LIN {X 0,Y 181.648,Z 836.947,A -85,B 0,C 180,E1 -22430.375,E2 -22430.375} C_VEL
LIN {X 0,Y 184.597,Z 832.968,A -85,B 0,C 180,E1 -22433.56,E2 -22433.56} C_VEL
LIN {X 0,Y 188.035,Z 827.945,A -85,B 0,C 180,E1 -22436.645,E2 -22436.645} C_VEL
LIN {X 0,Y 192.221,Z 821.754,A -85,B 0,C 180,E1 -22439.574,E2 -22439.574} C_VEL
LIN {X 0,Y 196.99,Z 814.161,A -85,B 0,C 180,E1 -22442.351,E2 -22442.351} C_VEL
LIN {X 0,Y 201.347,Z 806.526,A -85,B 0,C 180,E1 -22444.553,E2 -22444.553} C_VEL
LIN {X 0,Y 206.537,Z 796.463,A -85,B 0,C 180,E1 -22446.848,E2 -22446.848} C_VEL
LIN {X 0,Y 211.759,Z 785.133,A -85,B 0,C 180,E1 -22448.785,E2 -22448.785} C_VEL
LIN {X 0,Y 216.158,Z 773.945,A -85,B 0,C 180,E1 -22450.253,E2 -22450.253} C_VEL
LIN {X 0,Y 220.233,Z 761.427,A -85,B 0,C 180,E1 -22451.462,E2 -22451.462} C_VEL
LIN {X 0,Y 223.58,Z 747.939,A -85,B 0,C 180,E1 -22452.442,E2 -22452.442} C_VEL
LIN {X 0,Y 226.11,Z 733.339,A -85,B 0,C 180,E1 -22453.139,E2 -22453.139} C_VEL
LIN {X 0,Y 229.571,Z 702.946,A -85,B 0,C 180,E1 -22454.32,E2 -22454.32} C_VEL
LIN {X 0,Y 229.531,Z 699.375,A -85,B 0,C 180,E1 -22454.67,E2 -22454.67} C_VEL
LIN {X 0,Y 226.994,Z 691.679,A -85,B 0,C 180,E1 -22456.697,E2 -22456.697} C_VEL
LIN {X 0,Y 224.698,Z 685.638,A -85,B 0,C 180,E1 -22458.748,E2 -22458.748} C_VEL
LIN {X 0,Y 223.199,Z 682.051,A -85,B 0,C 180,E1 -22460.219,E2 -22460.219} C_VEL
LIN {X 0,Y 221.344,Z 677.62,A -85,B 0,C 180,E1 -22462.368,E2 -22462.368} C_VEL
LIN {X 0,Y 219.109,Z 672.518,A -85,B 0,C 180,E1 -22465.767,E2 -22465.767} C_VEL
LIN {X 0,Y 217.682,Z 669.713,A -85,B 0,C 180,E1 -22469.18,E2 -22469.18} C_VEL
LIN {X 0,Y 217.221,Z 667.959,A -85,B 0,C 180,E1 -22473.066,E2 -22473.066} C_VEL
LIN {X 0,Y 217.771,Z 667.973,A -85,B 0,C 180,E1 -22476.348,E2 -22476.348} C_VEL
LIN {X 0,Y 219.129,Z 668.973,A -85,B 0,C 180,E1 -22479.449,E2 -22479.449} C_VEL
LIN {X 0,Y 221.964,Z 672.987,A -85,B 0,C 180,E1 -22483.528,E2 -22483.528} C_VEL
LIN {X 0,Y 224.726,Z 677.151,A -85,B 0,C 180,E1 -22486.32,E2 -22486.32} C_VEL
LIN {X 0,Y 226.55,Z 680.51,A -85,B 0,C 180,E1 -22487.887,E2 -22487.887} C_VEL
LIN {X 0,Y 230.041,Z 686.961,A -85,B 0,C 180,E1 -22490.49,E2 -22490.49} C_VEL
LIN {X 0,Y 230.883,Z 688.932,A -85,B 0,C 180,E1 -22491.084,E2 -22491.084} C_VEL
LIN {X 0,Y 226.569,Z 725.397,A -85,B 0,C 180,E1 -22492.505,E2 -22492.505} C_VEL
LIN {X 0,Y 224.368,Z 737.74,A -85,B 0,C 180,E1 -22493.254,E2 -22493.254} C_VEL
LIN {X 0,Y 221.212,Z 750.989,A -85,B 0,C 180,E1 -22494.416,E2 -22494.416} C_VEL
LIN {X 0,Y 217.435,Z 762.949,A -85,B 0,C 180,E1 -22495.805,E2 -22495.805} C_VEL
LIN {X 0,Y 212.855,Z 774.862,A -85,B 0,C 180,E1 -22497.634,E2 -22497.634} C_VEL
LIN {X 0,Y 208.036,Z 785.272,A -85,B 0,C 180,E1 -22499.74,E2 -22499.74} C_VEL
LIN {X 0,Y 203.356,Z 793.978,A -85,B 0,C 180,E1 -22501.98,E2 -22501.98} C_VEL
LIN {X 0,Y 198.482,Z 801.986,A -85,B 0,C 180,E1 -22504.581,E2 -22504.581} C_VEL
LIN {X 0,Y 193.325,Z 809.445,A -85,B 0,C 180,E1 -22507.835,E2 -22507.835} C_VEL
LIN {X 0,Y 189.546,Z 814.354,A -85,B 0,C 180,E1 -22510.684,E2 -22510.684} C_VEL
LIN {X 0,Y 185.596,Z 818.913,A -85,B 0,C 180,E1 -22514.249,E2 -22514.249} C_VEL
LIN {X 0,Y 182.384,Z 822.122,A -85,B 0,C 180,E1 -22517.955,E2 -22517.955} C_VEL
LIN {X 0,Y 180.43,Z 823.653,A -85,B 0,C 180,E1 -22520.807,E2 -22520.807} C_VEL
LIN {X 0,Y 178.282,Z 824.713,A -85,B 0,C 180,E1 -22524.957,E2 -22524.957} C_VEL
LIN {X 0,Y 176.87,Z 824.404,A -85,B 0,C 180,E1 -22529.058,E2 -22529.058} C_VEL
LIN {X 0,Y 176.148,Z 822.83,A -85,B 0,C 180,E1 -22533.09,E2 -22533.09} C_VEL
LIN {X 0,Y 176.035,Z 820.076,A -85,B 0,C 180,E1 -22537.02,E2 -22537.02} C_VEL
LIN {X 0,Y 176.43,Z 816.179,A -85,B 0,C 180,E1 -22540.816,E2 -22540.816} C_VEL
LIN {X 0,Y 177.181,Z 811.17,A -85,B 0,C 180,E1 -22544.444,E2 -22544.444} C_VEL
LIN {X 0,Y 178.243,Z 804.98,A -85,B 0,C 180,E1 -22547.914,E2 -22547.914} C_VEL
LIN {X 0,Y 179.786,Z 796.986,A -85,B 0,C 180,E1 -22551.427,E2 -22551.427} C_VEL
LIN {X 0,Y 181.615,Z 788.148,A -85,B 0,C 180,E1 -22554.52,E2 -22554.52} C_VEL
LIN {X 0,Y 183.659,Z 777.988,A -85,B 0,C 180,E1 -22557.337,E2 -22557.337} C_VEL
LIN {X 0,Y 185.886,Z 766.319,A -85,B 0,C 180,E1 -22559.898,E2 -22559.898} C_VEL
LIN {X 0,Y 187.769,Z 754.884,A -85,B 0,C 180,E1 -22561.85,E2 -22561.85} C_VEL
LIN {X 0,Y 189.687,Z 741.422,A -85,B 0,C 180,E1 -22563.605,E2 -22563.605} C_VEL
LIN {X 0,Y 191.005,Z 727.938,A -85,B 0,C 180,E1 -22564.867,E2 -22564.867} C_VEL
LIN {X 0,Y 192.045,Z 714.44,A -85,B 0,C 180,E1 -22565.695,E2 -22565.695} C_VEL
LIN {X 0,Y 195.016,Z 662.361,A -85,B 0,C 180,E1 -22568.021,E2 -22568.021} C_VEL
LIN {X 0,Y 186.643,Z 641.655,A -85,B 0,C 180,E1 -22570.193,E2 -22570.193} C_VEL
LIN {X 0,Y 178.912,Z 624.29,A -85,B 0,C 180,E1 -22572.279,E2 -22572.279} C_VEL
LIN {X 0,Y 178.686,Z 623.228,A -85,B 0,C 180,E1 -22572.403,E2 -22572.403} C_VEL
LIN {X 0,Y 178.894,Z 623.2,A -85,B 0,C 180,E1 -22579.156,E2 -22579.156} C_VEL
LIN {X 0,Y 178.935,Z 623.197,A -85,B 0,C 180,E1 -22583.236,E2 -22583.236} C_VEL
LIN {X 0,Y 179.156,Z 623.169,A -85,B 0,C 180,E1 -22587.754,E2 -22587.754} C_VEL
LIN {X 0,Y 179.371,Z 623.142,A -85,B 0,C 180,E1 -22590.002,E2 -22590.002} C_VEL
LIN {X 0,Y 178.881,Z 623.204,A -85,B 0,C 180,E1 -22594.509,E2 -22594.509} C_VEL
LIN {X 0,Y 178.98,Z 623.19,A -85,B 0,C 180,E1 -22599.039,E2 -22599.039} C_VEL
LIN {X 0,Y 178.684,Z 623.226,A -85,B 0,C 180,E1 -22603.652,E2 -22603.652} C_VEL
LIN {X 0,Y 178.626,Z 623.218,A -85,B 0,C 180,E1 -22609.219,E2 -22609.219} C_VEL
LIN {X 0,Y 178.538,Z 623.247,A -85,B 0,C 180,E1 -22615.127,E2 -22615.127} C_VEL
LIN {X 0,Y 178.505,Z 623.239,A -85,B 0,C 180,E1 -22620.788,E2 -22620.788} C_VEL
LIN {X 0,Y 178.489,Z 623.223,A -85,B 0,C 180,E1 -22624.221,E2 -22624.221} C_VEL
LIN {X 0,Y 178.4,Z 623.256,A -85,B 0,C 180,E1 -22629.076,E2 -22629.076} C_VEL
LIN {X 0,Y 178.412,Z 623.258,A -85,B 0,C 180,E1 -22632.044,E2 -22632.044} C_VEL
LIN {X 0,Y 178.4,Z 623.259,A -85,B 0,C 180,E1 -22635.165,E2 -22635.165} C_VEL
LIN {X 0,Y 178.409,Z 623.246,A -85,B 0,C 180,E1 -22638.461,E2 -22638.461} C_VEL
LIN {X 0,Y 178.428,Z 623.228,A -85,B 0,C 180,E1 -22643.785,E2 -22643.785} C_VEL
LIN {X 0,Y 178.493,Z 623.236,A -85,B 0,C 180,E1 -22646.548,E2 -22646.548} C_VEL
LIN {X 0,Y 178.529,Z 623.245,A -85,B 0,C 180,E1 -22650.008,E2 -22650.008} C_VEL
LIN {X 0,Y 178.526,Z 623.245,A -85,B 0,C 180,E1 -22654.887,E2 -22654.887} C_VEL
LIN {X 0,Y 178.628,Z 623.214,A -85,B 0,C 180,E1 -22660.787,E2 -22660.787} C_VEL
LIN {X 0,Y 178.663,Z 623.21,A -85,B 0,C 180,E1 -22666.349,E2 -22666.349} C_VEL
LIN {X 0,Y 178.919,Z 623.194,A -85,B 0,C 180,E1 -22670.96,E2 -22670.96} C_VEL
LIN {X 0,Y 179.159,Z 623.161,A -85,B 0,C 180,E1 -22677.752,E2 -22677.752} C_VEL
LIN {X 0,Y 179.377,Z 623.123,A -85,B 0,C 180,E1 -22680,E2 -22680} C_VEL
LIN {X 0,Y 178.874,Z 623.193,A -85,B 0,C 180,E1 -22684.507,E2 -22684.507} C_VEL
LIN {X 0,Y 178.919,Z 623.197,A -85,B 0,C 180,E1 -22689.04,E2 -22689.04} C_VEL
LIN {X 0,Y 178.653,Z 623.223,A -85,B 0,C 180,E1 -22693.653,E2 -22693.653} C_VEL
LIN {X 0,Y 178.597,Z 623.239,A -85,B 0,C 180,E1 -22699.185,E2 -22699.185} C_VEL
LIN {X 0,Y 178.527,Z 623.24,A -85,B 0,C 180,E1 -22705.114,E2 -22705.114} C_VEL
LIN {X 0,Y 178.508,Z 623.25,A -85,B 0,C 180,E1 -22710.786,E2 -22710.786} C_VEL
LIN {X 0,Y 178.492,Z 623.248,A -85,B 0,C 180,E1 -22714.219,E2 -22714.219} C_VEL
LIN {X 0,Y 178.402,Z 623.264,A -85,B 0,C 180,E1 -22719.073,E2 -22719.073} C_VEL
LIN {X 0,Y 178.405,Z 623.264,A -85,B 0,C 180,E1 -22722.044,E2 -22722.044} C_VEL
LIN {X 0,Y 178.457,Z 623.395,A -85,B 0,C 180,E1 -22727.484,E2 -22727.484} C_VEL
LIN {X 0,Y 180.474,Z 632.149,A -85,B 0,C 180,E1 -22732.051,E2 -22732.051} C_VEL
LIN {X 0,Y 180.651,Z 633.055,A -85,B 0,C 180,E1 -22732.32,E2 -22732.32} C_VEL
LIN {X 0,Y 188.835,Z 656.224,A -85,B 0,C 180,E1 -22734.741,E2 -22734.741} C_VEL
LIN {X 0,Y 190.706,Z 662.523,A -85,B 0,C 180,E1 -22735.314,E2 -22735.314} C_VEL
LIN {X 0,Y 193.865,Z 696.157,A -85,B 0,C 180,E1 -22737.428,E2 -22737.428} C_VEL
LIN {X 0,Y 191.64,Z 736.563,A -85,B 0,C 180,E1 -22739.265,E2 -22739.265} C_VEL
LIN {X 0,Y 190.442,Z 742.309,A -85,B 0,C 180,E1 -22739.495,E2 -22739.495} C_VEL
LIN {X 0,Y 186.806,Z 751.468,A -85,B 0,C 180,E1 -22739.876,E2 -22739.876} C_VEL
LIN {X 0,Y 183.032,Z 760.446,A -85,B 0,C 180,E1 -22740.48,E2 -22740.48} C_VEL
LIN {X 0,Y 181.66,Z 765.908,A -85,B 0,C 180,E1 -22741.063,E2 -22741.063} C_VEL
LIN {X 0,Y 179.478,Z 778.762,A -85,B 0,C 180,E1 -22742.919,E2 -22742.919} C_VEL
LIN {X 0,Y 177.326,Z 790.159,A -85,B 0,C 180,E1 -22745.093,E2 -22745.093} C_VEL
LIN {X 0,Y 175.234,Z 800.711,A -85,B 0,C 180,E1 -22747.649,E2 -22747.649} C_VEL
LIN {X 0,Y 173.269,Z 809.87,A -85,B 0,C 180,E1 -22750.447,E2 -22750.447} C_VEL
LIN {X 0,Y 171.502,Z 818.953,A -85,B 0,C 180,E1 -22753.94,E2 -22753.94} C_VEL
LIN {X 0,Y 170.239,Z 826.179,A -85,B 0,C 180,E1 -22757.48,E2 -22757.48} C_VEL
LIN {X 0,Y 169.735,Z 831.058,A -85,B 0,C 180,E1 -22760.464,E2 -22760.464} C_VEL
LIN {X 0,Y 169.564,Z 835.798,A -85,B 0,C 180,E1 -22764.125,E2 -22764.125} C_VEL
LIN {X 0,Y 169.464,Z 839.133,A -85,B 0,C 180,E1 -22767.621,E2 -22767.621} C_VEL
LIN {X 0,Y 169.461,Z 840.784,A -85,B 0,C 180,E1 -22769.997,E2 -22769.997} C_VEL
LIN {X 0,Y 169.352,Z 841.973,A -85,B 0,C 180,E1 -22772.376,E2 -22772.376} C_VEL
LIN {X 0,Y 169.192,Z 842.737,A -85,B 0,C 180,E1 -22774.763,E2 -22774.763} C_VEL
LIN {X 0,Y 169.156,Z 843.105,A -85,B 0,C 180,E1 -22777.157,E2 -22777.157} C_VEL
LIN {X 0,Y 169.944,Z 842.621,A -85,B 0,C 180,E1 -22781.931,E2 -22781.931} C_VEL
LIN {X 0,Y 171.776,Z 840.625,A -85,B 0,C 180,E1 -22786.64,E2 -22786.64} C_VEL
LIN {X 0,Y 174.132,Z 838.085,A -85,B 0,C 180,E1 -22790.061,E2 -22790.061} C_VEL
LIN {X 0,Y 176.987,Z 834.626,A -85,B 0,C 180,E1 -22793.394,E2 -22793.394} C_VEL
LIN {X 0,Y 180.46,Z 830.184,A -85,B 0,C 180,E1 -22796.603,E2 -22796.603} C_VEL
LIN {X 0,Y 185.371,Z 823.582,A -85,B 0,C 180,E1 -22800.153,E2 -22800.153} C_VEL
LIN {X 0,Y 191.098,Z 815.187,A -85,B 0,C 180,E1 -22803.478,E2 -22803.478} C_VEL
LIN {X 0,Y 196.603,Z 806.297,A -85,B 0,C 180,E1 -22806.142,E2 -22806.142} C_VEL
LIN {X 0,Y 202.055,Z 796.335,A -85,B 0,C 180,E1 -22808.44,E2 -22808.44} C_VEL
LIN {X 0,Y 207.512,Z 785.05,A -85,B 0,C 180,E1 -22810.367,E2 -22810.367} C_VEL
LIN {X 0,Y 212.688,Z 772.449,A -85,B 0,C 180,E1 -22811.997,E2 -22811.997} C_VEL
LIN {X 0,Y 216.916,Z 759.806,A -85,B 0,C 180,E1 -22813.189,E2 -22813.189} C_VEL
LIN {X 0,Y 220.294,Z 746.746,A -85,B 0,C 180,E1 -22814.094,E2 -22814.094} C_VEL
LIN {X 0,Y 222.866,Z 732.04,A -85,B 0,C 180,E1 -22814.787,E2 -22814.787} C_VEL
LIN {X 0,Y 226.152,Z 704.076,A -85,B 0,C 180,E1 -22815.88,E2 -22815.88} C_VEL
LIN {X 0,Y 225.993,Z 702.661,A -85,B 0,C 180,E1 -22816.101,E2 -22816.101} C_VEL
LIN {X 0,Y 223.948,Z 695.907,A -85,B 0,C 180,E1 -22818.012,E2 -22818.012} C_VEL
LIN {X 0,Y 222.056,Z 690.697,A -85,B 0,C 180,E1 -22819.879,E2 -22819.879} C_VEL
LIN {X 0,Y 219.717,Z 684.472,A -85,B 0,C 180,E1 -22822.696,E2 -22822.696} C_VEL
LIN {X 0,Y 217.5,Z 679.143,A -85,B 0,C 180,E1 -22826.322,E2 -22826.322} C_VEL
LIN {X 0,Y 216.338,Z 676.59,A -85,B 0,C 180,E1 -22829.469,E2 -22829.469} C_VEL
LIN {X 0,Y 215.981,Z 675.016,A -85,B 0,C 180,E1 -22832.899,E2 -22832.899} C_VEL
LIN {X 0,Y 216.492,Z 674.945,A -85,B 0,C 180,E1 -22836.2,E2 -22836.2} C_VEL
LIN {X 0,Y 217.744,Z 675.898,A -85,B 0,C 180,E1 -22839.204,E2 -22839.204} C_VEL
LIN {X 0,Y 220.248,Z 679.639,A -85,B 0,C 180,E1 -22843.065,E2 -22843.065} C_VEL
LIN {X 0,Y 222.809,Z 683.707,A -85,B 0,C 180,E1 -22845.803,E2 -22845.803} C_VEL
LIN {X 0,Y 225.856,Z 689.7,A -85,B 0,C 180,E1 -22848.516,E2 -22848.516} C_VEL
LIN {X 0,Y 227.222,Z 692.457,A -85,B 0,C 180,E1 -22849.602,E2 -22849.602} C_VEL
LIN {X 0,Y 223.019,Z 726.729,A -85,B 0,C 180,E1 -22850.976,E2 -22850.976} C_VEL
LIN {X 0,Y 220.819,Z 738.383,A -85,B 0,C 180,E1 -22851.679,E2 -22851.679} C_VEL
LIN {X 0,Y 217.6,Z 751.285,A -85,B 0,C 180,E1 -22852.81,E2 -22852.81} C_VEL
LIN {X 0,Y 213.823,Z 762.651,A -85,B 0,C 180,E1 -22854.104,E2 -22854.104} C_VEL
LIN {X 0,Y 208.991,Z 774.646,A -85,B 0,C 180,E1 -22855.933,E2 -22855.933} C_VEL
LIN {X 0,Y 204.693,Z 783.723,A -85,B 0,C 180,E1 -22857.689,E2 -22857.689} C_VEL
LIN {X 0,Y 199.568,Z 793.055,A -85,B 0,C 180,E1 -22860,E2 -22860} C_VEL
LIN {X 0,Y 194.308,Z 801.252,A -85,B 0,C 180,E1 -22862.591,E2 -22862.591} C_VEL
LIN {X 0,Y 189.33,Z 808.21,A -85,B 0,C 180,E1 -22865.49,E2 -22865.49} C_VEL
LIN {X 0,Y 184.548,Z 814.138,A -85,B 0,C 180,E1 -22868.762,E2 -22868.762} C_VEL
LIN {X 0,Y 179.974,Z 819.021,A -85,B 0,C 180,E1 -22872.525,E2 -22872.525} C_VEL
LIN {X 0,Y 176.113,Z 822.597,A -85,B 0,C 180,E1 -22876.725,E2 -22876.725} C_VEL
LIN {X 0,Y 173.136,Z 824.6,A -85,B 0,C 180,E1 -22881.001,E2 -22881.001} C_VEL
LIN {X 0,Y 171.005,Z 825.207,A -85,B 0,C 180,E1 -22885.296,E2 -22885.296} C_VEL
LIN {X 0,Y 169.568,Z 824.435,A -85,B 0,C 180,E1 -22889.825,E2 -22889.825} C_VEL
LIN {X 0,Y 168.995,Z 822.592,A -85,B 0,C 180,E1 -22893.727,E2 -22893.727} C_VEL
LIN {X 0,Y 169.023,Z 819.432,A -85,B 0,C 180,E1 -22897.817,E2 -22897.817} C_VEL
LIN {X 0,Y 169.48,Z 815.16,A -85,B 0,C 180,E1 -22901.723,E2 -22901.723} C_VEL
LIN {X 0,Y 170.325,Z 809.758,A -85,B 0,C 180,E1 -22905.46,E2 -22905.46} C_VEL
LIN {X 0,Y 171.522,Z 803.165,A -85,B 0,C 180,E1 -22909.039,E2 -22909.039} C_VEL
LIN {X 0,Y 173.146,Z 795.104,A -85,B 0,C 180,E1 -22912.497,E2 -22912.497} C_VEL
LIN {X 0,Y 175.254,Z 785.219,A -85,B 0,C 180,E1 -22915.849,E2 -22915.849} C_VEL
LIN {X 0,Y 177.249,Z 775.473,A -85,B 0,C 180,E1 -22918.483,E2 -22918.483} C_VEL
LIN {X 0,Y 179.643,Z 763.151,A -85,B 0,C 180,E1 -22921.086,E2 -22921.086} C_VEL
LIN {X 0,Y 181.482,Z 751.827,A -85,B 0,C 180,E1 -22922.96,E2 -22922.96} C_VEL
LIN {X 0,Y 183.261,Z 738.622,A -85,B 0,C 180,E1 -22924.596,E2 -22924.596} C_VEL
LIN {X 0,Y 184.585,Z 724.922,A -85,B 0,C 180,E1 -22925.816,E2 -22925.816} C_VEL
LIN {X 0,Y 185.73,Z 707.38,A -85,B 0,C 180,E1 -22926.761,E2 -22926.761} C_VEL
LIN {X 0,Y 188.344,Z 663.896,A -85,B 0,C 180,E1 -22928.766,E2 -22928.766} C_VEL
LIN {X 0,Y 180.387,Z 644.222,A -85,B 0,C 180,E1 -22930.922,E2 -22930.922} C_VEL
LIN {X 0,Y 172.266,Z 626.336,A -85,B 0,C 180,E1 -22933.199,E2 -22933.199} C_VEL
LIN {X 0,Y 171.62,Z 624.104,A -85,B 0,C 180,E1 -22933.498,E2 -22933.498} C_VEL
LIN {X 0,Y 171.84,Z 624.079,A -85,B 0,C 180,E1 -22938.98,E2 -22938.98} C_VEL
LIN {X 0,Y 171.9,Z 624.074,A -85,B 0,C 180,E1 -22942.957,E2 -22942.957} C_VEL
LIN {X 0,Y 172.103,Z 624.048,A -85,B 0,C 180,E1 -22947.662,E2 -22947.662} C_VEL
LIN {X 0,Y 172.334,Z 624.019,A -85,B 0,C 180,E1 -22950.003,E2 -22950.003} C_VEL
LIN {X 0,Y 171.83,Z 624.083,A -85,B 0,C 180,E1 -22954.695,E2 -22954.695} C_VEL
LIN {X 0,Y 171.912,Z 624.07,A -85,B 0,C 180,E1 -22959.414,E2 -22959.414} C_VEL
LIN {X 0,Y 171.597,Z 624.109,A -85,B 0,C 180,E1 -22964.228,E2 -22964.228} C_VEL
LIN {X 0,Y 171.547,Z 624.098,A -85,B 0,C 180,E1 -22969.564,E2 -22969.564} C_VEL
LIN {X 0,Y 171.473,Z 624.125,A -85,B 0,C 180,E1 -22975.619,E2 -22975.619} C_VEL
LIN {X 0,Y 171.462,Z 624.117,A -85,B 0,C 180,E1 -22980.598,E2 -22980.598} C_VEL
LIN {X 0,Y 171.397,Z 624.109,A -85,B 0,C 180,E1 -22985.037,E2 -22985.037} C_VEL
LIN {X 0,Y 171.362,Z 624.131,A -85,B 0,C 180,E1 -22988.809,E2 -22988.809} C_VEL
LIN {X 0,Y 171.328,Z 624.139,A -85,B 0,C 180,E1 -22994.218,E2 -22994.218} C_VEL
LIN {X 0,Y 171.341,Z 624.123,A -85,B 0,C 180,E1 -22998.983,E2 -22998.983} C_VEL
LIN {X 0,Y 171.392,Z 624.097,A -85,B 0,C 180,E1 -23002.042,E2 -23002.042} C_VEL
LIN {X 0,Y 171.404,Z 624.11,A -85,B 0,C 180,E1 -23005.094,E2 -23005.094} C_VEL
LIN {X 0,Y 171.455,Z 624.124,A -85,B 0,C 180,E1 -23010.536,E2 -23010.536} C_VEL
LIN {X 0,Y 171.451,Z 624.125,A -85,B 0,C 180,E1 -23015.801,E2 -23015.801} C_VEL
LIN {X 0,Y 171.584,Z 624.09,A -85,B 0,C 180,E1 -23020.872,E2 -23020.872} C_VEL
LIN {X 0,Y 171.581,Z 624.087,A -85,B 0,C 180,E1 -23025.773,E2 -23025.773} C_VEL
LIN {X 0,Y 171.855,Z 624.074,A -85,B 0,C 180,E1 -23030.586,E2 -23030.586} C_VEL
LIN {X 0,Y 171.822,Z 624.079,A -85,B 0,C 180,E1 -23035.308,E2 -23035.308} C_VEL
LIN {X 0,Y 172.34,Z 623.998,A -85,B 0,C 180,E1 -23040,E2 -23040} C_VEL
LIN {X 0,Y 171.822,Z 624.072,A -85,B 0,C 180,E1 -23044.693,E2 -23044.693} C_VEL
LIN {X 0,Y 171.856,Z 624.077,A -85,B 0,C 180,E1 -23049.415,E2 -23049.415} C_VEL
LIN {X 0,Y 171.567,Z 624.102,A -85,B 0,C 180,E1 -23054.228,E2 -23054.228} C_VEL
LIN {X 0,Y 171.522,Z 624.12,A -85,B 0,C 180,E1 -23059.533,E2 -23059.533} C_VEL
LIN {X 0,Y 171.466,Z 624.12,A -85,B 0,C 180,E1 -23065.609,E2 -23065.609} C_VEL
LIN {X 0,Y 171.466,Z 624.129,A -85,B 0,C 180,E1 -23070.595,E2 -23070.595} C_VEL
LIN {X 0,Y 171.4,Z 624.136,A -85,B 0,C 180,E1 -23075.034,E2 -23075.034} C_VEL
LIN {X 0,Y 171.364,Z 624.142,A -85,B 0,C 180,E1 -23078.806,E2 -23078.806} C_VEL
LIN {X 0,Y 171.328,Z 624.146,A -85,B 0,C 180,E1 -23084.216,E2 -23084.216} C_VEL
LIN {X 0,Y 171.392,Z 624.272,A -85,B 0,C 180,E1 -23086.817,E2 -23086.817} C_VEL
LIN {X 0,Y 173.24,Z 632.25,A -85,B 0,C 180,E1 -23091.139,E2 -23091.139} C_VEL
LIN {X 0,Y 181.647,Z 655.872,A -85,B 0,C 180,E1 -23093.752,E2 -23093.752} C_VEL
LIN {X 0,Y 184.297,Z 664.633,A -85,B 0,C 180,E1 -23094.603,E2 -23094.603} C_VEL
LIN {X 0,Y 187.221,Z 696.409,A -85,B 0,C 180,E1 -23096.685,E2 -23096.685} C_VEL
LIN {X 0,Y 184.484,Z 742.136,A -85,B 0,C 180,E1 -23098.888,E2 -23098.888} C_VEL
LIN {X 0,Y 183.189,Z 755.342,A -85,B 0,C 180,E1 -23099.922,E2 -23099.922} C_VEL
LIN {X 0,Y 181.66,Z 765.908,A -85,B 0,C 180,E1 -23101.063,E2 -23101.063} C_VEL
LIN {X 0,Y 180.156,Z 771.254,A -85,B 0,C 180,E1 -23101.703,E2 -23101.703} C_VEL
LIN {X 0,Y 175.928,Z 779.57,A -85,B 0,C 180,E1 -23102.786,E2 -23102.786} C_VEL
LIN {X 0,Y 171.556,Z 787.511,A -85,B 0,C 180,E1 -23104.131,E2 -23104.131} C_VEL
LIN {X 0,Y 169.855,Z 792.272,A -85,B 0,C 180,E1 -23105.168,E2 -23105.168} C_VEL
LIN {X 0,Y 167.776,Z 802.309,A -85,B 0,C 180,E1 -23107.849,E2 -23107.849} C_VEL
LIN {X 0,Y 165.879,Z 811.256,A -85,B 0,C 180,E1 -23110.828,E2 -23110.828} C_VEL
LIN {X 0,Y 164.405,Z 818.635,A -85,B 0,C 180,E1 -23113.865,E2 -23113.865} C_VEL
LIN {X 0,Y 163.159,Z 825.839,A -85,B 0,C 180,E1 -23117.56,E2 -23117.56} C_VEL
LIN {X 0,Y 162.576,Z 831.543,A -85,B 0,C 180,E1 -23121.295,E2 -23121.295} C_VEL
LIN {X 0,Y 162.512,Z 835.963,A -85,B 0,C 180,E1 -23125.035,E2 -23125.035} C_VEL
LIN {X 0,Y 162.41,Z 838.219,A -85,B 0,C 180,E1 -23127.517,E2 -23127.517} C_VEL
LIN {X 0,Y 162.397,Z 840.008,A -85,B 0,C 180,E1 -23129.997,E2 -23129.997} C_VEL
LIN {X 0,Y 162.285,Z 841.286,A -85,B 0,C 180,E1 -23132.479,E2 -23132.479} C_VEL
LIN {X 0,Y 162.126,Z 842.116,A -85,B 0,C 180,E1 -23134.971,E2 -23134.971} C_VEL
LIN {X 0,Y 162.396,Z 842.622,A -85,B 0,C 180,E1 -23139.966,E2 -23139.966} C_VEL
LIN {X 0,Y 162.953,Z 842.305,A -85,B 0,C 180,E1 -23142.451,E2 -23142.451} C_VEL
LIN {X 0,Y 164.975,Z 840.477,A -85,B 0,C 180,E1 -23147.347,E2 -23147.347} C_VEL
LIN {X 0,Y 168.35,Z 837.157,A -85,B 0,C 180,E1 -23152.066,E2 -23152.066} C_VEL
LIN {X 0,Y 172.082,Z 833.095,A -85,B 0,C 180,E1 -23155.837,E2 -23155.837} C_VEL
LIN {X 0,Y 176.954,Z 827.175,A -85,B 0,C 180,E1 -23159.763,E2 -23159.763} C_VEL
LIN {X 0,Y 182.672,Z 819.937,A -85,B 0,C 180,E1 -23163.244,E2 -23163.244} C_VEL
LIN {X 0,Y 188.074,Z 812.235,A -85,B 0,C 180,E1 -23166.051,E2 -23166.051} C_VEL
LIN {X 0,Y 194.06,Z 802.72,A -85,B 0,C 180,E1 -23168.658,E2 -23168.658} C_VEL
LIN {X 0,Y 198.865,Z 794.219,A -85,B 0,C 180,E1 -23170.492,E2 -23170.492} C_VEL
LIN {X 0,Y 204.672,Z 782.701,A -85,B 0,C 180,E1 -23172.364,E2 -23172.364} C_VEL
LIN {X 0,Y 209.455,Z 771.196,A -85,B 0,C 180,E1 -23173.789,E2 -23173.789} C_VEL
LIN {X 0,Y 214.151,Z 757.338,A -85,B 0,C 180,E1 -23175.04,E2 -23175.04} C_VEL
LIN {X 0,Y 217.473,Z 744.314,A -85,B 0,C 180,E1 -23175.863,E2 -23175.863} C_VEL
LIN {X 0,Y 219.913,Z 730.436,A -85,B 0,C 180,E1 -23176.497,E2 -23176.497} C_VEL
LIN {X 0,Y 222.876,Z 706.643,A -85,B 0,C 180,E1 -23177.423,E2 -23177.423} C_VEL
LIN {X 0,Y 220.939,Z 700.117,A -85,B 0,C 180,E1 -23179.419,E2 -23179.419} C_VEL
LIN {X 0,Y 219.165,Z 694.647,A -85,B 0,C 180,E1 -23181.566,E2 -23181.566} C_VEL
LIN {X 0,Y 217.607,Z 690.255,A -85,B 0,C 180,E1 -23183.771,E2 -23183.771} C_VEL
LIN {X 0,Y 216.016,Z 685.879,A -85,B 0,C 180,E1 -23186.782,E2 -23186.782} C_VEL
LIN {X 0,Y 214.98,Z 683.376,A -85,B 0,C 180,E1 -23189.928,E2 -23189.928} C_VEL
LIN {X 0,Y 214.743,Z 682.061,A -85,B 0,C 180,E1 -23192.73,E2 -23192.73} C_VEL
LIN {X 0,Y 215.228,Z 681.921,A -85,B 0,C 180,E1 -23196.102,E2 -23196.102} C_VEL
LIN {X 0,Y 216.338,Z 682.759,A -85,B 0,C 180,E1 -23198.895,E2 -23198.895} C_VEL
LIN {X 0,Y 218.64,Z 686.47,A -85,B 0,C 180,E1 -23202.692,E2 -23202.692} C_VEL
LIN {X 0,Y 220.809,Z 690.081,A -85,B 0,C 180,E1 -23205.176,E2 -23205.176} C_VEL
LIN {X 0,Y 223.856,Z 696.508,A -85,B 0,C 180,E1 -23208.093,E2 -23208.093} C_VEL
LIN {X 0,Y 219.867,Z 727.125,A -85,B 0,C 180,E1 -23209.329,E2 -23209.329} C_VEL
LIN {X 0,Y 217.502,Z 739.038,A -85,B 0,C 180,E1 -23210.054,E2 -23210.054} C_VEL
LIN {X 0,Y 214.344,Z 750.993,A -85,B 0,C 180,E1 -23211.084,E2 -23211.084} C_VEL
LIN {X 0,Y 210.603,Z 762.175,A -85,B 0,C 180,E1 -23212.329,E2 -23212.329} C_VEL
LIN {X 0,Y 206.193,Z 772.889,A -85,B 0,C 180,E1 -23213.885,E2 -23213.885} C_VEL
LIN {X 0,Y 200.639,Z 784.1,A -85,B 0,C 180,E1 -23215.983,E2 -23215.983} C_VEL
LIN {X 0,Y 194.872,Z 793.942,A -85,B 0,C 180,E1 -23218.45,E2 -23218.45} C_VEL
LIN {X 0,Y 189.768,Z 801.5,A -85,B 0,C 180,E1 -23220.853,E2 -23220.853} C_VEL
LIN {X 0,Y 184.358,Z 808.629,A -85,B 0,C 180,E1 -23223.825,E2 -23223.825} C_VEL
LIN {X 0,Y 179.771,Z 813.92,A -85,B 0,C 180,E1 -23226.735,E2 -23226.735} C_VEL
LIN {X 0,Y 174.938,Z 818.831,A -85,B 0,C 180,E1 -23230.415,E2 -23230.415} C_VEL
LIN {X 0,Y 170.911,Z 822.338,A -85,B 0,C 180,E1 -23234.283,E2 -23234.283} C_VEL
LIN {X 0,Y 168.679,Z 823.974,A -85,B 0,C 180,E1 -23236.957,E2 -23236.957} C_VEL
LIN {X 0,Y 165.824,Z 825.432,A -85,B 0,C 180,E1 -23241.195,E2 -23241.195} C_VEL
LIN {X 0,Y 163.71,Z 825.596,A -85,B 0,C 180,E1 -23245.648,E2 -23245.648} C_VEL
LIN {X 0,Y 162.396,Z 824.488,A -85,B 0,C 180,E1 -23250.062,E2 -23250.062} C_VEL
LIN {X 0,Y 161.862,Z 822.164,A -85,B 0,C 180,E1 -23254.419,E2 -23254.419} C_VEL
LIN {X 0,Y 161.995,Z 818.668,A -85,B 0,C 180,E1 -23258.66,E2 -23258.66} C_VEL
LIN {X 0,Y 162.574,Z 814.032,A -85,B 0,C 180,E1 -23262.705,E2 -23262.705} C_VEL
LIN {X 0,Y 163.632,Z 807.638,A -85,B 0,C 180,E1 -23266.898,E2 -23266.898} C_VEL
LIN {X 0,Y 164.863,Z 801.169,A -85,B 0,C 180,E1 -23270.254,E2 -23270.254} C_VEL
LIN {X 0,Y 166.691,Z 792.582,A -85,B 0,C 180,E1 -23273.828,E2 -23273.828} C_VEL
LIN {X 0,Y 168.726,Z 783.205,A -85,B 0,C 180,E1 -23276.914,E2 -23276.914} C_VEL
LIN {X 0,Y 170.929,Z 772.602,A -85,B 0,C 180,E1 -23279.705,E2 -23279.705} C_VEL
LIN {X 0,Y 172.995,Z 762.142,A -85,B 0,C 180,E1 -23281.893,E2 -23281.893} C_VEL
LIN {X 0,Y 175.074,Z 749.382,A -85,B 0,C 180,E1 -23283.966,E2 -23283.966} C_VEL
LIN {X 0,Y 176.713,Z 737.201,A -85,B 0,C 180,E1 -23285.461,E2 -23285.461} C_VEL
LIN {X 0,Y 177.996,Z 723.969,A -85,B 0,C 180,E1 -23286.617,E2 -23286.617} C_VEL
LIN {X 0,Y 179.405,Z 703.191,A -85,B 0,C 180,E1 -23287.729,E2 -23287.729} C_VEL
LIN {X 0,Y 181.754,Z 665.678,A -85,B 0,C 180,E1 -23289.525,E2 -23289.525} C_VEL
LIN {X 0,Y 174.275,Z 647.102,A -85,B 0,C 180,E1 -23291.639,E2 -23291.639} C_VEL
LIN {X 0,Y 165.654,Z 627.903,A -85,B 0,C 180,E1 -23294.192,E2 -23294.192} C_VEL
LIN {X 0,Y 164.569,Z 624.982,A -85,B 0,C 180,E1 -23294.601,E2 -23294.601} C_VEL
LIN {X 0,Y 164.85,Z 624.951,A -85,B 0,C 180,E1 -23300.184,E2 -23300.184} C_VEL
LIN {X 0,Y 164.862,Z 624.951,A -85,B 0,C 180,E1 -23302.655,E2 -23302.655} C_VEL
LIN {X 0,Y 165.052,Z 624.926,A -85,B 0,C 180,E1 -23307.562,E2 -23307.562} C_VEL
LIN {X 0,Y 165.297,Z 624.895,A -85,B 0,C 180,E1 -23310.003,E2 -23310.003} C_VEL
LIN {X 0,Y 164.78,Z 624.96,A -85,B 0,C 180,E1 -23314.896,E2 -23314.896} C_VEL
LIN {X 0,Y 164.855,Z 624.949,A -85,B 0,C 180,E1 -23319.821,E2 -23319.821} C_VEL
LIN {X 0,Y 164.539,Z 624.989,A -85,B 0,C 180,E1 -23324.852,E2 -23324.852} C_VEL
LIN {X 0,Y 164.476,Z 624.978,A -85,B 0,C 180,E1 -23329.991,E2 -23329.991} C_VEL
LIN {X 0,Y 164.397,Z 625.006,A -85,B 0,C 180,E1 -23336.136,E2 -23336.136} C_VEL
LIN {X 0,Y 164.392,Z 624.992,A -85,B 0,C 180,E1 -23341.238,E2 -23341.238} C_VEL
LIN {X 0,Y 164.299,Z 625.003,A -85,B 0,C 180,E1 -23346.791,E2 -23346.791} C_VEL
LIN {X 0,Y 164.296,Z 625.015,A -85,B 0,C 180,E1 -23349.918,E2 -23349.918} C_VEL
LIN {X 0,Y 164.284,Z 625.02,A -85,B 0,C 180,E1 -23353.344,E2 -23353.344} C_VEL
LIN {X 0,Y 164.297,Z 625.011,A -85,B 0,C 180,E1 -23356.811,E2 -23356.811} C_VEL
LIN {X 0,Y 164.3,Z 624.992,A -85,B 0,C 180,E1 -23360.354,E2 -23360.354} C_VEL
LIN {X 0,Y 164.336,Z 624.985,A -85,B 0,C 180,E1 -23364.351,E2 -23364.351} C_VEL
LIN {X 0,Y 164.397,Z 625,A -85,B 0,C 180,E1 -23369.136,E2 -23369.136} C_VEL
LIN {X 0,Y 164.413,Z 625.003,A -85,B 0,C 180,E1 -23374.694,E2 -23374.694} C_VEL
LIN {X 0,Y 164.491,Z 624.975,A -85,B 0,C 180,E1 -23380.053,E2 -23380.053} C_VEL
LIN {X 0,Y 164.511,Z 624.964,A -85,B 0,C 180,E1 -23385.148,E2 -23385.148} C_VEL
LIN {X 0,Y 164.775,Z 624.955,A -85,B 0,C 180,E1 -23390.177,E2 -23390.177} C_VEL
LIN {X 0,Y 164.838,Z 624.95,A -85,B 0,C 180,E1 -23392.652,E2 -23392.652} C_VEL
LIN {X 0,Y 165.055,Z 624.918,A -85,B 0,C 180,E1 -23397.56,E2 -23397.56} C_VEL
LIN {X 0,Y 165.302,Z 624.874,A -85,B 0,C 180,E1 -23400,E2 -23400} C_VEL
LIN {X 0,Y 164.771,Z 624.951,A -85,B 0,C 180,E1 -23404.894,E2 -23404.894} C_VEL
LIN {X 0,Y 164.839,Z 624.949,A -85,B 0,C 180,E1 -23407.349,E2 -23407.349} C_VEL
LIN {X 0,Y 164.71,Z 624.965,A -85,B 0,C 180,E1 -23411.061,E2 -23411.061} C_VEL
LIN {X 0,Y 164.46,Z 624.995,A -85,B 0,C 180,E1 -23417.406,E2 -23417.406} C_VEL
LIN {X 0,Y 164.456,Z 625.001,A -85,B 0,C 180,E1 -23419.992,E2 -23419.992} C_VEL
LIN {X 0,Y 164.393,Z 625.001,A -85,B 0,C 180,E1 -23426.128,E2 -23426.128} C_VEL
LIN {X 0,Y 164.396,Z 625.006,A -85,B 0,C 180,E1 -23431.235,E2 -23431.235} C_VEL
LIN {X 0,Y 164.301,Z 625.019,A -85,B 0,C 180,E1 -23436.788,E2 -23436.788} C_VEL
LIN {X 0,Y 164.297,Z 625.021,A -85,B 0,C 180,E1 -23439.915,E2 -23439.915} C_VEL
LIN {X 0,Y 164.288,Z 625.024,A -85,B 0,C 180,E1 -23444.897,E2 -23444.897} C_VEL
LIN {X 0,Y 164.337,Z 625.089,A -85,B 0,C 180,E1 -23446.082,E2 -23446.082} C_VEL
LIN {X 0,Y 165.907,Z 631.794,A -85,B 0,C 180,E1 -23449.914,E2 -23449.914} C_VEL
LIN {X 0,Y 174.901,Z 656.794,A -85,B 0,C 180,E1 -23452.854,E2 -23452.854} C_VEL
LIN {X 0,Y 177.785,Z 665.671,A -85,B 0,C 180,E1 -23453.773,E2 -23453.773} C_VEL
LIN {X 0,Y 180.611,Z 696.413,A -85,B 0,C 180,E1 -23455.882,E2 -23455.882} C_VEL
LIN {X 0,Y 177.779,Z 741.96,A -85,B 0,C 180,E1 -23458.16,E2 -23458.16} C_VEL
LIN {X 0,Y 176.362,Z 755.741,A -85,B 0,C 180,E1 -23459.295,E2 -23459.295} C_VEL
LIN {X 0,Y 174.452,Z 768.195,A -85,B 0,C 180,E1 -23460.757,E2 -23460.757} C_VEL
LIN {X 0,Y 172.23,Z 780.264,A -85,B 0,C 180,E1 -23462.67,E2 -23462.67} C_VEL
LIN {X 0,Y 170.078,Z 791.308,A -85,B 0,C 180,E1 -23464.938,E2 -23464.938} C_VEL
LIN {X 0,Y 169.855,Z 792.272,A -85,B 0,C 180,E1 -23465.168,E2 -23465.168} C_VEL
LIN {X 0,Y 168.17,Z 796.897,A -85,B 0,C 180,E1 -23466.293,E2 -23466.293} C_VEL
LIN {X 0,Y 163.831,Z 803.893,A -85,B 0,C 180,E1 -23468.206,E2 -23468.206} C_VEL
LIN {X 0,Y 159.597,Z 810.395,A -85,B 0,C 180,E1 -23470.404,E2 -23470.404} C_VEL
LIN {X 0,Y 158.11,Z 814.21,A -85,B 0,C 180,E1 -23471.939,E2 -23471.939} C_VEL
LIN {X 0,Y 156.601,Z 822.119,A -85,B 0,C 180,E1 -23475.707,E2 -23475.707} C_VEL
LIN {X 0,Y 155.719,Z 828.51,A -85,B 0,C 180,E1 -23479.597,E2 -23479.597} C_VEL
LIN {X 0,Y 155.439,Z 834.189,A -85,B 0,C 180,E1 -23484.107,E2 -23484.107} C_VEL
LIN {X 0,Y 155.359,Z 837.282,A -85,B 0,C 180,E1 -23487.404,E2 -23487.404} C_VEL
LIN {X 0,Y 155.342,Z 839.144,A -85,B 0,C 180,E1 -23489.997,E2 -23489.997} C_VEL
LIN {X 0,Y 155.22,Z 840.542,A -85,B 0,C 180,E1 -23492.592,E2 -23492.592} C_VEL
LIN {X 0,Y 155.046,Z 841.481,A -85,B 0,C 180,E1 -23495.199,E2 -23495.199} C_VEL
LIN {X 0,Y 155.388,Z 842.15,A -85,B 0,C 180,E1 -23500.42,E2 -23500.42} C_VEL
LIN {X 0,Y 156.87,Z 841.331,A -85,B 0,C 180,E1 -23505.59,E2 -23505.59} C_VEL
LIN {X 0,Y 159.879,Z 838.979,A -85,B 0,C 180,E1 -23510.586,E2 -23510.586} C_VEL
LIN {X 0,Y 164.048,Z 835.058,A -85,B 0,C 180,E1 -23515.364,E2 -23515.364} C_VEL
LIN {X 0,Y 167.907,Z 831.031,A -85,B 0,C 180,E1 -23518.77,E2 -23518.77} C_VEL
LIN {X 0,Y 172.46,Z 825.955,A -85,B 0,C 180,E1 -23521.987,E2 -23521.987} C_VEL
LIN {X 0,Y 178.589,Z 818.53,A -85,B 0,C 180,E1 -23525.479,E2 -23525.479} C_VEL
LIN {X 0,Y 184.463,Z 810.644,A -85,B 0,C 180,E1 -23528.249,E2 -23528.249} C_VEL
LIN {X 0,Y 190.857,Z 801.001,A -85,B 0,C 180,E1 -23530.811,E2 -23530.811} C_VEL
LIN {X 0,Y 196.599,Z 791.168,A -85,B 0,C 180,E1 -23532.779,E2 -23532.779} C_VEL
LIN {X 0,Y 202.675,Z 778.963,A -85,B 0,C 180,E1 -23534.6,E2 -23534.6} C_VEL
LIN {X 0,Y 207.748,Z 766.798,A -85,B 0,C 180,E1 -23535.958,E2 -23535.958} C_VEL
LIN {X 0,Y 212.093,Z 753.545,A -85,B 0,C 180,E1 -23537.034,E2 -23537.034} C_VEL
LIN {X 0,Y 215.479,Z 739.849,A -85,B 0,C 180,E1 -23537.803,E2 -23537.803} C_VEL
LIN {X 0,Y 218.315,Z 720.921,A -85,B 0,C 180,E1 -23538.564,E2 -23538.564} C_VEL
LIN {X 0,Y 219.717,Z 709.868,A -85,B 0,C 180,E1 -23539.011,E2 -23539.011} C_VEL
LIN {X 0,Y 217.893,Z 703.232,A -85,B 0,C 180,E1 -23541.3,E2 -23541.3} C_VEL
LIN {X 0,Y 216.639,Z 699.413,A -85,B 0,C 180,E1 -23543.019,E2 -23543.019} C_VEL
LIN {X 0,Y 215.773,Z 696.529,A -85,B 0,C 180,E1 -23544.543,E2 -23544.543} C_VEL
LIN {X 0,Y 214.526,Z 692.552,A -85,B 0,C 180,E1 -23547.294,E2 -23547.294} C_VEL
LIN {X 0,Y 213.681,Z 690.279,A -85,B 0,C 180,E1 -23550.205,E2 -23550.205} C_VEL
LIN {X 0,Y 213.522,Z 688.933,A -85,B 0,C 180,E1 -23553.444,E2 -23553.444} C_VEL
LIN {X 0,Y 214.318,Z 689.078,A -85,B 0,C 180,E1 -23557.134,E2 -23557.134} C_VEL
LIN {X 0,Y 215.11,Z 690.06,A -85,B 0,C 180,E1 -23559.046,E2 -23559.046} C_VEL
LIN {X 0,Y 216.943,Z 693.058,A -85,B 0,C 180,E1 -23562.164,E2 -23562.164} C_VEL
LIN {X 0,Y 218.934,Z 696.625,A -85,B 0,C 180,E1 -23564.645,E2 -23564.645} C_VEL
LIN {X 0,Y 220.653,Z 700.602,A -85,B 0,C 180,E1 -23566.545,E2 -23566.545} C_VEL
LIN {X 0,Y 216.893,Z 728.131,A -85,B 0,C 180,E1 -23567.662,E2 -23567.662} C_VEL
LIN {X 0,Y 214.085,Z 741.371,A -85,B 0,C 180,E1 -23568.479,E2 -23568.479} C_VEL
LIN {X 0,Y 210.655,Z 753.344,A -85,B 0,C 180,E1 -23569.548,E2 -23569.548} C_VEL
LIN {X 0,Y 206.43,Z 764.7,A -85,B 0,C 180,E1 -23570.849,E2 -23570.849} C_VEL
LIN {X 0,Y 201.637,Z 775.401,A -85,B 0,C 180,E1 -23572.475,E2 -23572.475} C_VEL
LIN {X 0,Y 195.817,Z 786.26,A -85,B 0,C 180,E1 -23574.594,E2 -23574.594} C_VEL
LIN {X 0,Y 190.01,Z 795.516,A -85,B 0,C 180,E1 -23576.986,E2 -23576.986} C_VEL
LIN {X 0,Y 184.54,Z 802.988,A -85,B 0,C 180,E1 -23579.454,E2 -23579.454} C_VEL
LIN {X 0,Y 179.236,Z 809.433,A -85,B 0,C 180,E1 -23582.247,E2 -23582.247} C_VEL
LIN {X 0,Y 173.438,Z 815.572,A -85,B 0,C 180,E1 -23585.814,E2 -23585.814} C_VEL
LIN {X 0,Y 168.396,Z 820.168,A -85,B 0,C 180,E1 -23589.61,E2 -23589.61} C_VEL
LIN {X 0,Y 165.43,Z 822.504,A -85,B 0,C 180,E1 -23592.295,E2 -23592.295} C_VEL
LIN {X 0,Y 161.508,Z 825.003,A -85,B 0,C 180,E1 -23596.809,E2 -23596.809} C_VEL
LIN {X 0,Y 158.506,Z 826.1,A -85,B 0,C 180,E1 -23601.398,E2 -23601.398} C_VEL
LIN {X 0,Y 156.422,Z 825.868,A -85,B 0,C 180,E1 -23606.033,E2 -23606.033} C_VEL
LIN {X 0,Y 155.181,Z 824.351,A -85,B 0,C 180,E1 -23610.634,E2 -23610.634} C_VEL
LIN {X 0,Y 154.759,Z 821.612,A -85,B 0,C 180,E1 -23615.178,E2 -23615.178} C_VEL
LIN {X 0,Y 154.963,Z 817.723,A -85,B 0,C 180,E1 -23619.561,E2 -23619.561} C_VEL
LIN {X 0,Y 155.709,Z 812.68,A -85,B 0,C 180,E1 -23623.771,E2 -23623.771} C_VEL
LIN {X 0,Y 156.776,Z 806.512,A -85,B 0,C 180,E1 -23627.75,E2 -23627.75} C_VEL
LIN {X 0,Y 158.281,Z 798.984,A -85,B 0,C 180,E1 -23631.569,E2 -23631.569} C_VEL
LIN {X 0,Y 160.332,Z 789.805,A -85,B 0,C 180,E1 -23635.264,E2 -23635.264} C_VEL
LIN {X 0,Y 162.446,Z 780.34,A -85,B 0,C 180,E1 -23638.279,E2 -23638.279} C_VEL
LIN {X 0,Y 164.688,Z 769.498,A -85,B 0,C 180,E1 -23641.024,E2 -23641.024} C_VEL
LIN {X 0,Y 167.005,Z 757.465,A -85,B 0,C 180,E1 -23643.412,E2 -23643.412} C_VEL
LIN {X 0,Y 169.004,Z 744.872,A -85,B 0,C 180,E1 -23645.304,E2 -23645.304} C_VEL
LIN {X 0,Y 170.651,Z 731.287,A -85,B 0,C 180,E1 -23646.811,E2 -23646.811} C_VEL
LIN {X 0,Y 171.868,Z 717.051,A -85,B 0,C 180,E1 -23647.84,E2 -23647.84} C_VEL
LIN {X 0,Y 175.082,Z 667.143,A -85,B 0,C 180,E1 -23650.34,E2 -23650.34} C_VEL
LIN {X 0,Y 166.978,Z 647.126,A -85,B 0,C 180,E1 -23652.775,E2 -23652.775} C_VEL
LIN {X 0,Y 158.692,Z 628.928,A -85,B 0,C 180,E1 -23655.366,E2 -23655.366} C_VEL
LIN {X 0,Y 157.651,Z 626.528,A -85,B 0,C 180,E1 -23655.721,E2 -23655.721} C_VEL
LIN {X 0,Y 157.538,Z 625.861,A -85,B 0,C 180,E1 -23655.801,E2 -23655.801} C_VEL
LIN {X 0,Y 157.768,Z 625.832,A -85,B 0,C 180,E1 -23659.739,E2 -23659.739} C_VEL
LIN {X 0,Y 157.824,Z 625.827,A -85,B 0,C 180,E1 -23662.326,E2 -23662.326} C_VEL
LIN {X 0,Y 158.259,Z 625.772,A -85,B 0,C 180,E1 -23670.003,E2 -23670.003} C_VEL
LIN {X 0,Y 157.827,Z 625.823,A -85,B 0,C 180,E1 -23677.68,E2 -23677.68} C_VEL
LIN {X 0,Y 157.707,Z 625.837,A -85,B 0,C 180,E1 -23681.364,E2 -23681.364} C_VEL
LIN {X 0,Y 157.465,Z 625.868,A -85,B 0,C 180,E1 -23685.536,E2 -23685.536} C_VEL
LIN {X 0,Y 157.373,Z 625.866,A -85,B 0,C 180,E1 -23690.935,E2 -23690.935} C_VEL
LIN {X 0,Y 157.319,Z 625.889,A -85,B 0,C 180,E1 -23696.688,E2 -23696.688} C_VEL
LIN {X 0,Y 157.285,Z 625.87,A -85,B 0,C 180,E1 -23702.428,E2 -23702.428} C_VEL
LIN {X 0,Y 157.272,Z 625.876,A -85,B 0,C 180,E1 -23706.452,E2 -23706.452} C_VEL
LIN {X 0,Y 157.215,Z 625.898,A -85,B 0,C 180,E1 -23712.113,E2 -23712.113} C_VEL
LIN {X 0,Y 157.216,Z 625.885,A -85,B 0,C 180,E1 -23717.891,E2 -23717.891} C_VEL
LIN {X 0,Y 157.273,Z 625.856,A -85,B 0,C 180,E1 -23723.552,E2 -23723.552} C_VEL
LIN {X 0,Y 157.3,Z 625.881,A -85,B 0,C 180,E1 -23728.097,E2 -23728.097} C_VEL
LIN {X 0,Y 157.322,Z 625.889,A -85,B 0,C 180,E1 -23733.466,E2 -23733.466} C_VEL
LIN {X 0,Y 157.398,Z 625.86,A -85,B 0,C 180,E1 -23739.671,E2 -23739.671} C_VEL
LIN {X 0,Y 157.447,Z 625.837,A -85,B 0,C 180,E1 -23744.466,E2 -23744.466} C_VEL
LIN {X 0,Y 157.697,Z 625.834,A -85,B 0,C 180,E1 -23749.732,E2 -23749.732} C_VEL
LIN {X 0,Y 157.775,Z 625.831,A -85,B 0,C 180,E1 -23752.321,E2 -23752.321} C_VEL
LIN {X 0,Y 158.265,Z 625.749,A -85,B 0,C 180,E1 -23760,E2 -23760} C_VEL
LIN {X 0,Y 157.775,Z 625.829,A -85,B 0,C 180,E1 -23767.68,E2 -23767.68} C_VEL
LIN {X 0,Y 157.641,Z 625.846,A -85,B 0,C 180,E1 -23771.23,E2 -23771.23} C_VEL
LIN {X 0,Y 157.429,Z 625.86,A -85,B 0,C 180,E1 -23775.537,E2 -23775.537} C_VEL
LIN {X 0,Y 157.364,Z 625.886,A -85,B 0,C 180,E1 -23780.934,E2 -23780.934} C_VEL
LIN {X 0,Y 157.316,Z 625.885,A -85,B 0,C 180,E1 -23786.68,E2 -23786.68} C_VEL
LIN {X 0,Y 157.288,Z 625.889,A -85,B 0,C 180,E1 -23792.425,E2 -23792.425} C_VEL
LIN {X 0,Y 157.275,Z 625.894,A -85,B 0,C 180,E1 -23796.448,E2 -23796.448} C_VEL
LIN {X 0,Y 157.217,Z 625.904,A -85,B 0,C 180,E1 -23802.109,E2 -23802.109} C_VEL
LIN {X 0,Y 157.281,Z 625.967,A -85,B 0,C 180,E1 -23805.35,E2 -23805.35} C_VEL
LIN {X 0,Y 158.497,Z 631.34,A -85,B 0,C 180,E1 -23808.576,E2 -23808.576} C_VEL
LIN {X 0,Y 166.387,Z 652.552,A -85,B 0,C 180,E1 -23811.299,E2 -23811.299} C_VEL
LIN {X 0,Y 171.371,Z 668.004,A -85,B 0,C 180,E1 -23813.013,E2 -23813.013} C_VEL
LIN {X 0,Y 173.975,Z 696.993,A -85,B 0,C 180,E1 -23815.084,E2 -23815.084} C_VEL
LIN {X 0,Y 171.123,Z 741.157,A -85,B 0,C 180,E1 -23817.379,E2 -23817.379} C_VEL
LIN {X 0,Y 169.734,Z 754.327,A -85,B 0,C 180,E1 -23818.48,E2 -23818.48} C_VEL
LIN {X 0,Y 167.95,Z 766.06,A -85,B 0,C 180,E1 -23819.855,E2 -23819.855} C_VEL
LIN {X 0,Y 165.669,Z 778.535,A -85,B 0,C 180,E1 -23821.837,E2 -23821.837} C_VEL
LIN {X 0,Y 163.403,Z 789.798,A -85,B 0,C 180,E1 -23824.181,E2 -23824.181} C_VEL
LIN {X 0,Y 161.207,Z 800.063,A -85,B 0,C 180,E1 -23826.895,E2 -23826.895} C_VEL
LIN {X 0,Y 159.154,Z 809.302,A -85,B 0,C 180,E1 -23829.985,E2 -23829.985} C_VEL
LIN {X 0,Y 158.11,Z 814.21,A -85,B 0,C 180,E1 -23831.939,E2 -23831.939} C_VEL
LIN {X 0,Y 156.689,Z 817.844,A -85,B 0,C 180,E1 -23833.559,E2 -23833.559} C_VEL
LIN {X 0,Y 152.862,Z 823.049,A -85,B 0,C 180,E1 -23836.347,E2 -23836.347} C_VEL
LIN {X 0,Y 149.356,Z 827.666,A -85,B 0,C 180,E1 -23839.425,E2 -23839.425} C_VEL
LIN {X 0,Y 148.465,Z 830.248,A -85,B 0,C 180,E1 -23841.441,E2 -23841.441} C_VEL
LIN {X 0,Y 148.379,Z 834.525,A -85,B 0,C 180,E1 -23845.272,E2 -23845.272} C_VEL
LIN {X 0,Y 148.31,Z 836.308,A -85,B 0,C 180,E1 -23847.281,E2 -23847.281} C_VEL
LIN {X 0,Y 148.288,Z 838.264,A -85,B 0,C 180,E1 -23849.997,E2 -23849.997} C_VEL
LIN {X 0,Y 148.067,Z 840.513,A -85,B 0,C 180,E1 -23854.605,E2 -23854.605} C_VEL
LIN {X 0,Y 148.007,Z 841.435,A -85,B 0,C 180,E1 -23858.187,E2 -23858.187} C_VEL
LIN {X 0,Y 149.034,Z 841.536,A -85,B 0,C 180,E1 -23863.635,E2 -23863.635} C_VEL
LIN {X 0,Y 151.444,Z 840.168,A -85,B 0,C 180,E1 -23868.953,E2 -23868.953} C_VEL
LIN {X 0,Y 155.253,Z 837.305,A -85,B 0,C 180,E1 -23874.039,E2 -23874.039} C_VEL
LIN {X 0,Y 160.304,Z 832.824,A -85,B 0,C 180,E1 -23878.83,E2 -23878.83} C_VEL
LIN {X 0,Y 164.831,Z 828.322,A -85,B 0,C 180,E1 -23882.203,E2 -23882.203} C_VEL
LIN {X 0,Y 171.089,Z 821.734,A -85,B 0,C 180,E1 -23885.825,E2 -23885.825} C_VEL
LIN {X 0,Y 176.963,Z 814.702,A -85,B 0,C 180,E1 -23888.716,E2 -23888.716} C_VEL
LIN {X 0,Y 183.408,Z 806.054,A -85,B 0,C 180,E1 -23891.373,E2 -23891.373} C_VEL
LIN {X 0,Y 189.129,Z 797.437,A -85,B 0,C 180,E1 -23893.426,E2 -23893.426} C_VEL
LIN {X 0,Y 195.294,Z 786.992,A -85,B 0,C 180,E1 -23895.292,E2 -23895.292} C_VEL
LIN {X 0,Y 201.042,Z 775.39,A -85,B 0,C 180,E1 -23896.862,E2 -23896.862} C_VEL
LIN {X 0,Y 205.733,Z 764.035,A -85,B 0,C 180,E1 -23897.984,E2 -23897.984} C_VEL
LIN {X 0,Y 209.903,Z 751.267,A -85,B 0,C 180,E1 -23898.957,E2 -23898.957} C_VEL
LIN {X 0,Y 213.219,Z 737.653,A -85,B 0,C 180,E1 -23899.674,E2 -23899.674} C_VEL
LIN {X 0,Y 216.764,Z 714.225,A -85,B 0,C 180,E1 -23900.567,E2 -23900.567} C_VEL
LIN {X 0,Y 216.803,Z 713.203,A -85,B 0,C 180,E1 -23900.685,E2 -23900.685} C_VEL
LIN {X 0,Y 215.285,Z 707.337,A -85,B 0,C 180,E1 -23902.917,E2 -23902.917} C_VEL
LIN {X 0,Y 214.082,Z 703.019,A -85,B 0,C 180,E1 -23905.152,E2 -23905.152} C_VEL
LIN {X 0,Y 213.063,Z 699.275,A -85,B 0,C 180,E1 -23907.762,E2 -23907.762} C_VEL
LIN {X 0,Y 212.375,Z 697.166,A -85,B 0,C 180,E1 -23910.511,E2 -23910.511} C_VEL
LIN {X 0,Y 212.26,Z 695.947,A -85,B 0,C 180,E1 -23913.372,E2 -23913.372} C_VEL
LIN {X 0,Y 212.88,Z 695.949,A -85,B 0,C 180,E1 -23916.661,E2 -23916.661} C_VEL
LIN {X 0,Y 213.651,Z 696.819,A -85,B 0,C 180,E1 -23918.617,E2 -23918.617} C_VEL
LIN {X 0,Y 215.342,Z 699.819,A -85,B 0,C 180,E1 -23921.753,E2 -23921.753} C_VEL
LIN {X 0,Y 217.094,Z 703.273,A -85,B 0,C 180,E1 -23924.141,E2 -23924.141} C_VEL
LIN {X 0,Y 217.769,Z 705.006,A -85,B 0,C 180,E1 -23924.964,E2 -23924.964} C_VEL
LIN {X 0,Y 214.289,Z 728.814,A -85,B 0,C 180,E1 -23925.919,E2 -23925.919} C_VEL
LIN {X 0,Y 211.456,Z 741.514,A -85,B 0,C 180,E1 -23926.691,E2 -23926.691} C_VEL
LIN {X 0,Y 208.202,Z 752.451,A -85,B 0,C 180,E1 -23927.625,E2 -23927.625} C_VEL
LIN {X 0,Y 203.405,Z 765.104,A -85,B 0,C 180,E1 -23929.045,E2 -23929.045} C_VEL
LIN {X 0,Y 197.877,Z 776.861,A -85,B 0,C 180,E1 -23930.802,E2 -23930.802} C_VEL
LIN {X 0,Y 192.009,Z 787.088,A -85,B 0,C 180,E1 -23932.817,E2 -23932.817} C_VEL
LIN {X 0,Y 186.07,Z 795.975,A -85,B 0,C 180,E1 -23935.125,E2 -23935.125} C_VEL
LIN {X 0,Y 179.917,Z 803.948,A -85,B 0,C 180,E1 -23937.761,E2 -23937.761} C_VEL
LIN {X 0,Y 173.216,Z 811.412,A -85,B 0,C 180,E1 -23941.162,E2 -23941.162} C_VEL
LIN {X 0,Y 167.163,Z 817.188,A -85,B 0,C 180,E1 -23944.823,E2 -23944.823} C_VEL
LIN {X 0,Y 161.816,Z 821.529,A -85,B 0,C 180,E1 -23948.782,E2 -23948.782} C_VEL
LIN {X 0,Y 157.462,Z 824.414,A -85,B 0,C 180,E1 -23952.895,E2 -23952.895} C_VEL
LIN {X 0,Y 154.181,Z 826.003,A -85,B 0,C 180,E1 -23956.827,E2 -23956.827} C_VEL
LIN {X 0,Y 151.06,Z 826.627,A -85,B 0,C 180,E1 -23961.851,E2 -23961.851} C_VEL
LIN {X 0,Y 149.13,Z 825.964,A -85,B 0,C 180,E1 -23966.447,E2 -23966.447} C_VEL
LIN {X 0,Y 147.935,Z 823.936,A -85,B 0,C 180,E1 -23971.505,E2 -23971.505} C_VEL
LIN {X 0,Y 147.669,Z 820.942,A -85,B 0,C 180,E1 -23976,E2 -23976} C_VEL
LIN {X 0,Y 148.003,Z 816.642,A -85,B 0,C 180,E1 -23980.561,E2 -23980.561} C_VEL
LIN {X 0,Y 148.901,Z 810.964,A -85,B 0,C 180,E1 -23985.071,E2 -23985.071} C_VEL
LIN {X 0,Y 150.062,Z 804.584,A -85,B 0,C 180,E1 -23989.033,E2 -23989.033} C_VEL
LIN {X 0,Y 151.766,Z 796.547,A -85,B 0,C 180,E1 -23992.99,E2 -23992.99} C_VEL
LIN {X 0,Y 154.07,Z 786.649,A -85,B 0,C 180,E1 -23996.816,E2 -23996.816} C_VEL
LIN {X 0,Y 156.224,Z 777.046,A -85,B 0,C 180,E1 -23999.769,E2 -23999.769} C_VEL
LIN {X 0,Y 158.571,Z 766.107,A -85,B 0,C 180,E1 -24002.426,E2 -24002.426} C_VEL
LIN {X 0,Y 160.714,Z 754.518,A -85,B 0,C 180,E1 -24004.645,E2 -24004.645} C_VEL
LIN {X 0,Y 162.653,Z 742.455,A -85,B 0,C 180,E1 -24006.412,E2 -24006.412} C_VEL
LIN {X 0,Y 164.254,Z 728.323,A -85,B 0,C 180,E1 -24007.907,E2 -24007.907} C_VEL
LIN {X 0,Y 165.4,Z 715.017,A -85,B 0,C 180,E1 -24008.812,E2 -24008.812} C_VEL
LIN {X 0,Y 168.446,Z 668.634,A -85,B 0,C 180,E1 -24011.218,E2 -24011.218} C_VEL
LIN {X 0,Y 160.781,Z 649.862,A -85,B 0,C 180,E1 -24013.611,E2 -24013.611} C_VEL
LIN {X 0,Y 153.53,Z 633.685,A -85,B 0,C 180,E1 -24016.013,E2 -24016.013} C_VEL
LIN {X 0,Y 150.664,Z 627.552,A -85,B 0,C 180,E1 -24017.005,E2 -24017.005} C_VEL
LIN {X 0,Y 150.545,Z 626.732,A -85,B 0,C 180,E1 -24017.144,E2 -24017.144} C_VEL
LIN {X 0,Y 150.762,Z 626.706,A -85,B 0,C 180,E1 -24021.964,E2 -24021.964} C_VEL
LIN {X 0,Y 151.22,Z 626.649,A -85,B 0,C 180,E1 -24030.003,E2 -24030.003} C_VEL
LIN {X 0,Y 150.765,Z 626.703,A -85,B 0,C 180,E1 -24038.042,E2 -24038.042} C_VEL
LIN {X 0,Y 150.637,Z 626.717,A -85,B 0,C 180,E1 -24041.548,E2 -24041.548} C_VEL
LIN {X 0,Y 150.371,Z 626.752,A -85,B 0,C 180,E1 -24046.289,E2 -24046.289} C_VEL
LIN {X 0,Y 150.354,Z 626.739,A -85,B 0,C 180,E1 -24050.795,E2 -24050.795} C_VEL
LIN {X 0,Y 150.249,Z 626.768,A -85,B 0,C 180,E1 -24057.286,E2 -24057.286} C_VEL
LIN {X 0,Y 150.224,Z 626.746,A -85,B 0,C 180,E1 -24062.638,E2 -24062.638} C_VEL
LIN {X 0,Y 150.177,Z 626.764,A -85,B 0,C 180,E1 -24067.476,E2 -24067.476} C_VEL
LIN {X 0,Y 150.155,Z 626.78,A -85,B 0,C 180,E1 -24071.507,E2 -24071.507} C_VEL
LIN {X 0,Y 150.13,Z 626.777,A -85,B 0,C 180,E1 -24075.397,E2 -24075.397} C_VEL
LIN {X 0,Y 150.155,Z 626.758,A -85,B 0,C 180,E1 -24079.06,E2 -24079.06} C_VEL
LIN {X 0,Y 150.184,Z 626.734,A -85,B 0,C 180,E1 -24082.71,E2 -24082.71} C_VEL
LIN {X 0,Y 150.221,Z 626.757,A -85,B 0,C 180,E1 -24087.369,E2 -24087.369} C_VEL
LIN {X 0,Y 150.247,Z 626.768,A -85,B 0,C 180,E1 -24092.722,E2 -24092.722} C_VEL
LIN {X 0,Y 150.356,Z 626.74,A -85,B 0,C 180,E1 -24099.211,E2 -24099.211} C_VEL
LIN {X 0,Y 150.358,Z 626.716,A -85,B 0,C 180,E1 -24103.713,E2 -24103.713} C_VEL
LIN {X 0,Y 150.618,Z 626.714,A -85,B 0,C 180,E1 -24109.243,E2 -24109.243} C_VEL
LIN {X 0,Y 150.712,Z 626.71,A -85,B 0,C 180,E1 -24111.959,E2 -24111.959} C_VEL
LIN {X 0,Y 151.225,Z 626.625,A -85,B 0,C 180,E1 -24120,E2 -24120} C_VEL
LIN {X 0,Y 150.712,Z 626.71,A -85,B 0,C 180,E1 -24128.042,E2 -24128.042} C_VEL
LIN {X 0,Y 150.583,Z 626.725,A -85,B 0,C 180,E1 -24131.433,E2 -24131.433} C_VEL
LIN {X 0,Y 150.337,Z 626.745,A -85,B 0,C 180,E1 -24136.29,E2 -24136.29} C_VEL
LIN {X 0,Y 150.346,Z 626.761,A -85,B 0,C 180,E1 -24140.779,E2 -24140.779} C_VEL
LIN {X 0,Y 150.249,Z 626.769,A -85,B 0,C 180,E1 -24147.279,E2 -24147.279} C_VEL
LIN {X 0,Y 150.227,Z 626.767,A -85,B 0,C 180,E1 -24152.634,E2 -24152.634} C_VEL
LIN {X 0,Y 150.179,Z 626.779,A -85,B 0,C 180,E1 -24157.472,E2 -24157.472} C_VEL
LIN {X 0,Y 150.161,Z 626.786,A -85,B 0,C 180,E1 -24162.915,E2 -24162.915} C_VEL
LIN {X 0,Y 150.225,Z 626.855,A -85,B 0,C 180,E1 -24164.568,E2 -24164.568} C_VEL
LIN {X 0,Y 151.159,Z 630.936,A -85,B 0,C 180,E1 -24167.141,E2 -24167.141} C_VEL
LIN {X 0,Y 158.261,Z 649.528,A -85,B 0,C 180,E1 -24169.753,E2 -24169.753} C_VEL
LIN {X 0,Y 164.951,Z 669.636,A -85,B 0,C 180,E1 -24172.145,E2 -24172.145} C_VEL
LIN {X 0,Y 167.292,Z 698.24,A -85,B 0,C 180,E1 -24174.261,E2 -24174.261} C_VEL
LIN {X 0,Y 164.399,Z 741.311,A -85,B 0,C 180,E1 -24176.603,E2 -24176.603} C_VEL
LIN {X 0,Y 162.965,Z 754.298,A -85,B 0,C 180,E1 -24177.742,E2 -24177.742} C_VEL
LIN {X 0,Y 161.15,Z 765.952,A -85,B 0,C 180,E1 -24179.171,E2 -24179.171} C_VEL
LIN {X 0,Y 158.789,Z 778.333,A -85,B 0,C 180,E1 -24181.225,E2 -24181.225} C_VEL
LIN {X 0,Y 156.469,Z 789.522,A -85,B 0,C 180,E1 -24183.655,E2 -24183.655} C_VEL
LIN {X 0,Y 154.194,Z 799.779,A -85,B 0,C 180,E1 -24186.493,E2 -24186.493} C_VEL
LIN {X 0,Y 152.108,Z 808.972,A -85,B 0,C 180,E1 -24189.722,E2 -24189.722} C_VEL
LIN {X 0,Y 150.258,Z 817.95,A -85,B 0,C 180,E1 -24193.699,E2 -24193.699} C_VEL
LIN {X 0,Y 148.984,Z 825.087,A -85,B 0,C 180,E1 -24197.741,E2 -24197.741} C_VEL
LIN {X 0,Y 148.465,Z 830.248,A -85,B 0,C 180,E1 -24201.441,E2 -24201.441} C_VEL
LIN {X 0,Y 147.683,Z 832.645,A -85,B 0,C 180,E1 -24203.508,E2 -24203.508} C_VEL
LIN {X 0,Y 146.064,Z 834.617,A -85,B 0,C 180,E1 -24205.605,E2 -24205.605} C_VEL
LIN {X 0,Y 142.323,Z 837.562,A -85,B 0,C 180,E1 -24210.007,E2 -24210.007} C_VEL
LIN {X 0,Y 141.075,Z 839.065,A -85,B 0,C 180,E1 -24213.161,E2 -24213.161} C_VEL
LIN {X 0,Y 140.973,Z 840.784,A -85,B 0,C 180,E1 -24218.598,E2 -24218.598} C_VEL
LIN {X 0,Y 142.116,Z 841.143,A -85,B 0,C 180,E1 -24224.312,E2 -24224.312} C_VEL
LIN {X 0,Y 144.72,Z 839.975,A -85,B 0,C 180,E1 -24229.87,E2 -24229.87} C_VEL
LIN {X 0,Y 148.792,Z 837.349,A -85,B 0,C 180,E1 -24235.154,E2 -24235.154} C_VEL
LIN {X 0,Y 153.259,Z 833.88,A -85,B 0,C 180,E1 -24239.391,E2 -24239.391} C_VEL
LIN {X 0,Y 158.9,Z 828.93,A -85,B 0,C 180,E1 -24243.56,E2 -24243.56} C_VEL
LIN {X 0,Y 165.442,Z 822.595,A -85,B 0,C 180,E1 -24247.25,E2 -24247.25} C_VEL
LIN {X 0,Y 171.563,Z 815.87,A -85,B 0,C 180,E1 -24250.176,E2 -24250.176} C_VEL
LIN {X 0,Y 178.25,Z 807.731,A -85,B 0,C 180,E1 -24252.85,E2 -24252.85} C_VEL
LIN {X 0,Y 184.168,Z 799.55,A -85,B 0,C 180,E1 -24254.905,E2 -24254.905} C_VEL
LIN {X 0,Y 190.507,Z 789.651,A -85,B 0,C 180,E1 -24256.765,E2 -24256.765} C_VEL
LIN {X 0,Y 197.071,Z 777.497,A -85,B 0,C 180,E1 -24258.492,E2 -24258.492} C_VEL
LIN {X 0,Y 202.59,Z 765.225,A -85,B 0,C 180,E1 -24259.743,E2 -24259.743} C_VEL
LIN {X 0,Y 207.105,Z 752.362,A -85,B 0,C 180,E1 -24260.722,E2 -24260.722} C_VEL
LIN {X 0,Y 210.611,Z 739.172,A -85,B 0,C 180,E1 -24261.425,E2 -24261.425} C_VEL
LIN {X 0,Y 213.665,Z 720.771,A -85,B 0,C 180,E1 -24262.128,E2 -24262.128} C_VEL
LIN {X 0,Y 214.165,Z 717.119,A -85,B 0,C 180,E1 -24262.283,E2 -24262.283} C_VEL
LIN {X 0,Y 213.154,Z 712.57,A -85,B 0,C 180,E1 -24264.185,E2 -24264.185} C_VEL
LIN {X 0,Y 212.227,Z 708.918,A -85,B 0,C 180,E1 -24266.168,E2 -24266.168} C_VEL
LIN {X 0,Y 211.581,Z 705.938,A -85,B 0,C 180,E1 -24268.328,E2 -24268.328} C_VEL
LIN {X 0,Y 211.061,Z 703.939,A -85,B 0,C 180,E1 -24271.004,E2 -24271.004} C_VEL
LIN {X 0,Y 211.09,Z 702.834,A -85,B 0,C 180,E1 -24274.013,E2 -24274.013} C_VEL
LIN {X 0,Y 211.98,Z 703.187,A -85,B 0,C 180,E1 -24277.578,E2 -24277.578} C_VEL
LIN {X 0,Y 213.677,Z 706.43,A -85,B 0,C 180,E1 -24281.219,E2 -24281.219} C_VEL
LIN {X 0,Y 215.035,Z 709.272,A -85,B 0,C 180,E1 -24283.289,E2 -24283.289} C_VEL
LIN {X 0,Y 211.767,Z 730.512,A -85,B 0,C 180,E1 -24284.184,E2 -24284.184} C_VEL
LIN {X 0,Y 208.902,Z 742.633,A -85,B 0,C 180,E1 -24284.913,E2 -24284.913} C_VEL
LIN {X 0,Y 205.303,Z 754.086,A -85,B 0,C 180,E1 -24285.887,E2 -24285.887} C_VEL
LIN {X 0,Y 200.629,Z 765.675,A -85,B 0,C 180,E1 -24287.18,E2 -24287.18} C_VEL
LIN {X 0,Y 194.93,Z 777.16,A -85,B 0,C 180,E1 -24288.868,E2 -24288.868} C_VEL
LIN {X 0,Y 188.647,Z 787.632,A -85,B 0,C 180,E1 -24290.89,E2 -24290.89} C_VEL
LIN {X 0,Y 181.964,Z 797.145,A -85,B 0,C 180,E1 -24293.346,E2 -24293.346} C_VEL
LIN {X 0,Y 175.459,Z 804.951,A -85,B 0,C 180,E1 -24295.979,E2 -24295.979} C_VEL
LIN {X 0,Y 168.678,Z 811.993,A -85,B 0,C 180,E1 -24299.243,E2 -24299.243} C_VEL
LIN {X 0,Y 162.957,Z 817.14,A -85,B 0,C 180,E1 -24302.471,E2 -24302.471} C_VEL
LIN {X 0,Y 157.42,Z 821.387,A -85,B 0,C 180,E1 -24306.211,E2 -24306.211} C_VEL
LIN {X 0,Y 152.166,Z 824.666,A -85,B 0,C 180,E1 -24310.646,E2 -24310.646} C_VEL
LIN {X 0,Y 149.398,Z 825.992,A -85,B 0,C 180,E1 -24313.604,E2 -24313.604} C_VEL
LIN {X 0,Y 146.854,Z 826.87,A -85,B 0,C 180,E1 -24316.847,E2 -24316.847} C_VEL
LIN {X 0,Y 143.856,Z 827.031,A -85,B 0,C 180,E1 -24321.848,E2 -24321.848} C_VEL
LIN {X 0,Y 141.832,Z 825.934,A -85,B 0,C 180,E1 -24326.891,E2 -24326.891} C_VEL
LIN {X 0,Y 140.765,Z 823.613,A -85,B 0,C 180,E1 -24331.929,E2 -24331.929} C_VEL
LIN {X 0,Y 140.606,Z 820.084,A -85,B 0,C 180,E1 -24336.901,E2 -24336.901} C_VEL
LIN {X 0,Y 141.08,Z 815.393,A -85,B 0,C 180,E1 -24341.654,E2 -24341.654} C_VEL
LIN {X 0,Y 142.049,Z 809.539,A -85,B 0,C 180,E1 -24346.164,E2 -24346.164} C_VEL
LIN {X 0,Y 143.423,Z 802.474,A -85,B 0,C 180,E1 -24350.434,E2 -24350.434} C_VEL
LIN {X 0,Y 145.347,Z 793.892,A -85,B 0,C 180,E1 -24354.537,E2 -24354.537} C_VEL
LIN {X 0,Y 147.626,Z 784.374,A -85,B 0,C 180,E1 -24358.109,E2 -24358.109} C_VEL
LIN {X 0,Y 150.152,Z 773.453,A -85,B 0,C 180,E1 -24361.355,E2 -24361.355} C_VEL
LIN {X 0,Y 152.546,Z 762.261,A -85,B 0,C 180,E1 -24363.947,E2 -24363.947} C_VEL
LIN {X 0,Y 154.794,Z 749.707,A -85,B 0,C 180,E1 -24366.196,E2 -24366.196} C_VEL
LIN {X 0,Y 156.754,Z 736.417,A -85,B 0,C 180,E1 -24367.95,E2 -24367.95} C_VEL
LIN {X 0,Y 158.206,Z 721.943,A -85,B 0,C 180,E1 -24369.272,E2 -24369.272} C_VEL
LIN {X 0,Y 161.916,Z 670.296,A -85,B 0,C 180,E1 -24372.099,E2 -24372.099} C_VEL
LIN {X 0,Y 152.539,Z 647.588,A -85,B 0,C 180,E1 -24375.23,E2 -24375.23} C_VEL
LIN {X 0,Y 143.774,Z 628.488,A -85,B 0,C 180,E1 -24378.37,E2 -24378.37} C_VEL
LIN {X 0,Y 143.618,Z 627.596,A -85,B 0,C 180,E1 -24378.536,E2 -24378.536} C_VEL
LIN {X 0,Y 143.683,Z 627.589,A -85,B 0,C 180,E1 -24381.565,E2 -24381.565} C_VEL
LIN {X 0,Y 144.178,Z 627.526,A -85,B 0,C 180,E1 -24390.003,E2 -24390.003} C_VEL
LIN {X 0,Y 143.687,Z 627.586,A -85,B 0,C 180,E1 -24398.441,E2 -24398.441} C_VEL
LIN {X 0,Y 143.573,Z 627.597,A -85,B 0,C 180,E1 -24401.761,E2 -24401.761} C_VEL
LIN {X 0,Y 143.308,Z 627.626,A -85,B 0,C 180,E1 -24407.115,E2 -24407.115} C_VEL
LIN {X 0,Y 143.28,Z 627.623,A -85,B 0,C 180,E1 -24411.257,E2 -24411.257} C_VEL
LIN {X 0,Y 143.196,Z 627.645,A -85,B 0,C 180,E1 -24417.941,E2 -24417.941} C_VEL
LIN {X 0,Y 143.151,Z 627.621,A -85,B 0,C 180,E1 -24423.425,E2 -24423.425} C_VEL
LIN {X 0,Y 143.066,Z 627.659,A -85,B 0,C 180,E1 -24429.692,E2 -24429.692} C_VEL
LIN {X 0,Y 143.061,Z 627.662,A -85,B 0,C 180,E1 -24433.457,E2 -24433.457} C_VEL
LIN {X 0,Y 143.07,Z 627.648,A -85,B 0,C 180,E1 -24437.467,E2 -24437.467} C_VEL
LIN {X 0,Y 143.082,Z 627.618,A -85,B 0,C 180,E1 -24441.808,E2 -24441.808} C_VEL
LIN {X 0,Y 143.188,Z 627.633,A -85,B 0,C 180,E1 -24447.323,E2 -24447.323} C_VEL
LIN {X 0,Y 143.195,Z 627.648,A -85,B 0,C 180,E1 -24452.066,E2 -24452.066} C_VEL
LIN {X 0,Y 143.281,Z 627.623,A -85,B 0,C 180,E1 -24458.749,E2 -24458.749} C_VEL
LIN {X 0,Y 143.301,Z 627.594,A -85,B 0,C 180,E1 -24462.887,E2 -24462.887} C_VEL
LIN {X 0,Y 143.544,Z 627.593,A -85,B 0,C 180,E1 -24468.706,E2 -24468.706} C_VEL
LIN {X 0,Y 143.633,Z 627.59,A -85,B 0,C 180,E1 -24471.559,E2 -24471.559} C_VEL
LIN {X 0,Y 144.184,Z 627.501,A -85,B 0,C 180,E1 -24480,E2 -24480} C_VEL
LIN {X 0,Y 143.633,Z 627.594,A -85,B 0,C 180,E1 -24488.441,E2 -24488.441} C_VEL
LIN {X 0,Y 143.509,Z 627.606,A -85,B 0,C 180,E1 -24491.621,E2 -24491.621} C_VEL
LIN {X 0,Y 143.276,Z 627.629,A -85,B 0,C 180,E1 -24497.117,E2 -24497.117} C_VEL
LIN {X 0,Y 143.274,Z 627.641,A -85,B 0,C 180,E1 -24501.244,E2 -24501.244} C_VEL
LIN {X 0,Y 143.197,Z 627.649,A -85,B 0,C 180,E1 -24507.936,E2 -24507.936} C_VEL
LIN {X 0,Y 143.154,Z 627.649,A -85,B 0,C 180,E1 -24513.421,E2 -24513.421} C_VEL
LIN {X 0,Y 143.067,Z 627.665,A -85,B 0,C 180,E1 -24519.689,E2 -24519.689} C_VEL
LIN {X 0,Y 143.14,Z 627.8,A -85,B 0,C 180,E1 -24523.788,E2 -24523.788} C_VEL
LIN {X 0,Y 143.74,Z 630.374,A -85,B 0,C 180,E1 -24525.525,E2 -24525.525} C_VEL
LIN {X 0,Y 150.931,Z 648.806,A -85,B 0,C 180,E1 -24528.373,E2 -24528.373} C_VEL
LIN {X 0,Y 157.854,Z 669.286,A -85,B 0,C 180,E1 -24530.998,E2 -24530.998} C_VEL
LIN {X 0,Y 158.581,Z 672.35,A -85,B 0,C 180,E1 -24531.318,E2 -24531.318} C_VEL
LIN {X 0,Y 160.684,Z 698.854,A -85,B 0,C 180,E1 -24533.356,E2 -24533.356} C_VEL
LIN {X 0,Y 157.722,Z 741.205,A -85,B 0,C 180,E1 -24535.764,E2 -24535.764} C_VEL
LIN {X 0,Y 156.228,Z 754.033,A -85,B 0,C 180,E1 -24536.941,E2 -24536.941} C_VEL
LIN {X 0,Y 154.374,Z 765.61,A -85,B 0,C 180,E1 -24538.426,E2 -24538.426} C_VEL
LIN {X 0,Y 151.95,Z 777.932,A -85,B 0,C 180,E1 -24540.562,E2 -24540.562} C_VEL
LIN {X 0,Y 149.344,Z 790.039,A -85,B 0,C 180,E1 -24543.336,E2 -24543.336} C_VEL
LIN {X 0,Y 147.225,Z 799.324,A -85,B 0,C 180,E1 -24546.058,E2 -24546.058} C_VEL
LIN {X 0,Y 145.071,Z 808.521,A -85,B 0,C 180,E1 -24549.435,E2 -24549.435} C_VEL
LIN {X 0,Y 143.166,Z 817.5,A -85,B 0,C 180,E1 -24553.601,E2 -24553.601} C_VEL
LIN {X 0,Y 141.911,Z 824.647,A -85,B 0,C 180,E1 -24557.847,E2 -24557.847} C_VEL
LIN {X 0,Y 141.368,Z 831.121,A -85,B 0,C 180,E1 -24562.859,E2 -24562.859} C_VEL
LIN {X 0,Y 141.264,Z 835.259,A -85,B 0,C 180,E1 -24567.145,E2 -24567.145} C_VEL
LIN {X 0,Y 141.236,Z 837.367,A -85,B 0,C 180,E1 -24569.997,E2 -24569.997} C_VEL
LIN {X 0,Y 141.075,Z 839.065,A -85,B 0,C 180,E1 -24573.161,E2 -24573.161} C_VEL
LIN {X 0,Y 140.306,Z 839.931,A -85,B 0,C 180,E1 -24575.518,E2 -24575.518} C_VEL
LIN {X 0,Y 137.607,Z 840.657,A -85,B 0,C 180,E1 -24579.441,E2 -24579.441} C_VEL
LIN {X 0,Y 135.71,Z 840.769,A -85,B 0,C 180,E1 -24582.694,E2 -24582.694} C_VEL
LIN {X 0,Y 135.358,Z 840.674,A -85,B 0,C 180,E1 -24585.202,E2 -24585.202} C_VEL
LIN {X 0,Y 135.566,Z 840.582,A -85,B 0,C 180,E1 -24586.034,E2 -24586.034} C_VEL
LIN {X 0,Y 138.042,Z 839.778,A -85,B 0,C 180,E1 -24590.875,E2 -24590.875} C_VEL
LIN {X 0,Y 142.392,Z 837.37,A -85,B 0,C 180,E1 -24596.369,E2 -24596.369} C_VEL
LIN {X 0,Y 148.026,Z 833.476,A -85,B 0,C 180,E1 -24601.48,E2 -24601.48} C_VEL
LIN {X 0,Y 153.057,Z 829.452,A -85,B 0,C 180,E1 -24605.024,E2 -24605.024} C_VEL
LIN {X 0,Y 158.899,Z 824.412,A -85,B 0,C 180,E1 -24608.255,E2 -24608.255} C_VEL
LIN {X 0,Y 165.178,Z 818.258,A -85,B 0,C 180,E1 -24611.257,E2 -24611.257} C_VEL
LIN {X 0,Y 172.023,Z 810.74,A -85,B 0,C 180,E1 -24613.986,E2 -24613.986} C_VEL
LIN {X 0,Y 179.326,Z 801.567,A -85,B 0,C 180,E1 -24616.468,E2 -24616.468} C_VEL
LIN {X 0,Y 186.512,Z 791.25,A -85,B 0,C 180,E1 -24618.492,E2 -24618.492} C_VEL
LIN {X 0,Y 193.285,Z 779.707,A -85,B 0,C 180,E1 -24620.182,E2 -24620.182} C_VEL
LIN {X 0,Y 198.931,Z 768.068,A -85,B 0,C 180,E1 -24621.408,E2 -24621.408} C_VEL
LIN {X 0,Y 203.932,Z 755.259,A -85,B 0,C 180,E1 -24622.428,E2 -24622.428} C_VEL
LIN {X 0,Y 207.928,Z 741.876,A -85,B 0,C 180,E1 -24623.152,E2 -24623.152} C_VEL
LIN {X 0,Y 210.819,Z 727.502,A -85,B 0,C 180,E1 -24623.745,E2 -24623.745} C_VEL
LIN {X 0,Y 211.791,Z 720.928,A -85,B 0,C 180,E1 -24624.002,E2 -24624.002} C_VEL
LIN {X 0,Y 210.802,Z 716.06,A -85,B 0,C 180,E1 -24626.386,E2 -24626.386} C_VEL
LIN {X 0,Y 210.104,Z 712.504,A -85,B 0,C 180,E1 -24628.982,E2 -24628.982} C_VEL
LIN {X 0,Y 209.76,Z 710.617,A -85,B 0,C 180,E1 -24631.628,E2 -24631.628} C_VEL
LIN {X 0,Y 209.862,Z 709.812,A -85,B 0,C 180,E1 -24634.192,E2 -24634.192} C_VEL
LIN {X 0,Y 210.657,Z 710.142,A -85,B 0,C 180,E1 -24637.43,E2 -24637.43} C_VEL
LIN {X 0,Y 212.009,Z 712.987,A -85,B 0,C 180,E1 -24640.64,E2 -24640.64} C_VEL
LIN {X 0,Y 212.595,Z 714.291,A -85,B 0,C 180,E1 -24641.637,E2 -24641.637} C_VEL
LIN {X 0,Y 209.595,Z 732.187,A -85,B 0,C 180,E1 -24642.391,E2 -24642.391} C_VEL
LIN {X 0,Y 206.528,Z 744.197,A -85,B 0,C 180,E1 -24643.119,E2 -24643.119} C_VEL
LIN {X 0,Y 202.475,Z 756.04,A -85,B 0,C 180,E1 -24644.136,E2 -24644.136} C_VEL
LIN {X 0,Y 197.077,Z 768.523,A -85,B 0,C 180,E1 -24645.544,E2 -24645.544} C_VEL
LIN {X 0,Y 191.023,Z 779.763,A -85,B 0,C 180,E1 -24647.247,E2 -24647.247} C_VEL
LIN {X 0,Y 184.356,Z 790.028,A -85,B 0,C 180,E1 -24649.289,E2 -24649.289} C_VEL
LIN {X 0,Y 177.568,Z 798.871,A -85,B 0,C 180,E1 -24651.662,E2 -24651.662} C_VEL
LIN {X 0,Y 169.999,Z 807.248,A -85,B 0,C 180,E1 -24654.618,E2 -24654.618} C_VEL
LIN {X 0,Y 163.721,Z 813.24,A -85,B 0,C 180,E1 -24657.539,E2 -24657.539} C_VEL
LIN {X 0,Y 156.879,Z 818.793,A -85,B 0,C 180,E1 -24661.283,E2 -24661.283} C_VEL
LIN {X 0,Y 150.763,Z 822.907,A -85,B 0,C 180,E1 -24665.349,E2 -24665.349} C_VEL
LIN {X 0,Y 147.192,Z 824.909,A -85,B 0,C 180,E1 -24668.235,E2 -24668.235} C_VEL
LIN {X 0,Y 143.569,Z 826.499,A -85,B 0,C 180,E1 -24671.767,E2 -24671.767} C_VEL
LIN {X 0,Y 139.513,Z 827.546,A -85,B 0,C 180,E1 -24676.85,E2 -24676.85} C_VEL
LIN {X 0,Y 136.517,Z 827.295,A -85,B 0,C 180,E1 -24682.091,E2 -24682.091} C_VEL
LIN {X 0,Y 134.555,Z 825.76,A -85,B 0,C 180,E1 -24687.393,E2 -24687.393} C_VEL
LIN {X 0,Y 133.59,Z 823.023,A -85,B 0,C 180,E1 -24692.682,E2 -24692.682} C_VEL
LIN {X 0,Y 133.567,Z 819.056,A -85,B 0,C 180,E1 -24697.889,E2 -24697.889} C_VEL
LIN {X 0,Y 134.186,Z 813.871,A -85,B 0,C 180,E1 -24702.912,E2 -24702.912} C_VEL
LIN {X 0,Y 135.273,Z 807.689,A -85,B 0,C 180,E1 -24707.519,E2 -24707.519} C_VEL
LIN {X 0,Y 136.887,Z 800.081,A -85,B 0,C 180,E1 -24711.973,E2 -24711.973} C_VEL
LIN {X 0,Y 139.087,Z 790.869,A -85,B 0,C 180,E1 -24716.237,E2 -24716.237} C_VEL
LIN {X 0,Y 141.622,Z 780.507,A -85,B 0,C 180,E1 -24719.972,E2 -24719.972} C_VEL
LIN {X 0,Y 144.181,Z 769.371,A -85,B 0,C 180,E1 -24723.118,E2 -24723.118} C_VEL
LIN {X 0,Y 146.609,Z 757.922,A -85,B 0,C 180,E1 -24725.616,E2 -24725.616} C_VEL
LIN {X 0,Y 148.902,Z 744.637,A -85,B 0,C 180,E1 -24727.819,E2 -24727.819} C_VEL
LIN {X 0,Y 150.679,Z 731.417,A -85,B 0,C 180,E1 -24729.396,E2 -24729.396} C_VEL
LIN {X 0,Y 152.002,Z 716.731,A -85,B 0,C 180,E1 -24730.555,E2 -24730.555} C_VEL
LIN {X 0,Y 155.281,Z 671.792,A -85,B 0,C 180,E1 -24733.072,E2 -24733.072} C_VEL
LIN {X 0,Y 146.33,Z 650.083,A -85,B 0,C 180,E1 -24736.241,E2 -24736.241} C_VEL
LIN {X 0,Y 137.683,Z 631.453,A -85,B 0,C 180,E1 -24739.526,E2 -24739.526} C_VEL
LIN {X 0,Y 136.576,Z 628.473,A -85,B 0,C 180,E1 -24740.095,E2 -24740.095} C_VEL
LIN {X 0,Y 136.757,Z 628.452,A -85,B 0,C 180,E1 -24747.057,E2 -24747.057} C_VEL
LIN {X 0,Y 137.136,Z 628.404,A -85,B 0,C 180,E1 -24750.003,E2 -24750.003} C_VEL
LIN {X 0,Y 136.61,Z 628.469,A -85,B 0,C 180,E1 -24758.881,E2 -24758.881} C_VEL
LIN {X 0,Y 136.494,Z 628.479,A -85,B 0,C 180,E1 -24761.959,E2 -24761.959} C_VEL
LIN {X 0,Y 136.247,Z 628.5,A -85,B 0,C 180,E1 -24768.032,E2 -24768.032} C_VEL
LIN {X 0,Y 136.201,Z 628.508,A -85,B 0,C 180,E1 -24771.752,E2 -24771.752} C_VEL
LIN {X 0,Y 136.122,Z 628.525,A -85,B 0,C 180,E1 -24778.633,E2 -24778.633} C_VEL
LIN {X 0,Y 136.048,Z 628.504,A -85,B 0,C 180,E1 -24784.631,E2 -24784.631} C_VEL
LIN {X 0,Y 136.036,Z 628.531,A -85,B 0,C 180,E1 -24789.201,E2 -24789.201} C_VEL
LIN {X 0,Y 136.002,Z 628.54,A -85,B 0,C 180,E1 -24793.66,E2 -24793.66} C_VEL
LIN {X 0,Y 136.01,Z 628.525,A -85,B 0,C 180,E1 -24797.798,E2 -24797.798} C_VEL
LIN {X 0,Y 136.031,Z 628.495,A -85,B 0,C 180,E1 -24801.686,E2 -24801.686} C_VEL
LIN {X 0,Y 136.091,Z 628.506,A -85,B 0,C 180,E1 -24805.723,E2 -24805.723} C_VEL
LIN {X 0,Y 136.151,Z 628.525,A -85,B 0,C 180,E1 -24812.318,E2 -24812.318} C_VEL
LIN {X 0,Y 136.248,Z 628.498,A -85,B 0,C 180,E1 -24818.834,E2 -24818.834} C_VEL
LIN {X 0,Y 136.27,Z 628.474,A -85,B 0,C 180,E1 -24825.057,E2 -24825.057} C_VEL
LIN {X 0,Y 136.438,Z 628.473,A -85,B 0,C 180,E1 -24828.167,E2 -24828.167} C_VEL
LIN {X 0,Y 136.559,Z 628.47,A -85,B 0,C 180,E1 -24831.119,E2 -24831.119} C_VEL
LIN {X 0,Y 137.141,Z 628.377,A -85,B 0,C 180,E1 -24840,E2 -24840} C_VEL
LIN {X 0,Y 136.558,Z 628.474,A -85,B 0,C 180,E1 -24848.882,E2 -24848.882} C_VEL
LIN {X 0,Y 136.423,Z 628.488,A -85,B 0,C 180,E1 -24851.892,E2 -24851.892} C_VEL
LIN {X 0,Y 136.195,Z 628.516,A -85,B 0,C 180,E1 -24858.036,E2 -24858.036} C_VEL
LIN {X 0,Y 136.197,Z 628.522,A -85,B 0,C 180,E1 -24861.739,E2 -24861.739} C_VEL
LIN {X 0,Y 136.124,Z 628.532,A -85,B 0,C 180,E1 -24868.628,E2 -24868.628} C_VEL
LIN {X 0,Y 136.051,Z 628.536,A -85,B 0,C 180,E1 -24874.627,E2 -24874.627} C_VEL
LIN {X 0,Y 136.038,Z 628.541,A -85,B 0,C 180,E1 -24879.197,E2 -24879.197} C_VEL
LIN {X 0,Y 136.088,Z 628.548,A -85,B 0,C 180,E1 -24882.811,E2 -24882.811} C_VEL
LIN {X 0,Y 136.373,Z 629.967,A -85,B 0,C 180,E1 -24883.818,E2 -24883.818} C_VEL
LIN {X 0,Y 143.917,Z 648.772,A -85,B 0,C 180,E1 -24886.976,E2 -24886.976} C_VEL
LIN {X 0,Y 151.069,Z 669.914,A -85,B 0,C 180,E1 -24889.885,E2 -24889.885} C_VEL
LIN {X 0,Y 152.175,Z 673.919,A -85,B 0,C 180,E1 -24890.358,E2 -24890.358} C_VEL
LIN {X 0,Y 154.161,Z 698.17,A -85,B 0,C 180,E1 -24892.339,E2 -24892.339} C_VEL
LIN {X 0,Y 151.074,Z 740.641,A -85,B 0,C 180,E1 -24894.849,E2 -24894.849} C_VEL
LIN {X 0,Y 149.54,Z 753.504,A -85,B 0,C 180,E1 -24896.073,E2 -24896.073} C_VEL
LIN {X 0,Y 147.63,Z 765.102,A -85,B 0,C 180,E1 -24897.615,E2 -24897.615} C_VEL
LIN {X 0,Y 145.146,Z 777.458,A -85,B 0,C 180,E1 -24899.841,E2 -24899.841} C_VEL
LIN {X 0,Y 142.696,Z 788.469,A -85,B 0,C 180,E1 -24902.441,E2 -24902.441} C_VEL
LIN {X 0,Y 140.251,Z 798.864,A -85,B 0,C 180,E1 -24905.578,E2 -24905.578} C_VEL
LIN {X 0,Y 138.023,Z 808.065,A -85,B 0,C 180,E1 -24909.115,E2 -24909.115} C_VEL
LIN {X 0,Y 136.093,Z 817.055,A -85,B 0,C 180,E1 -24913.496,E2 -24913.496} C_VEL
LIN {X 0,Y 134.836,Z 824.189,A -85,B 0,C 180,E1 -24917.963,E2 -24917.963} C_VEL
LIN {X 0,Y 134.326,Z 829.826,A -85,B 0,C 180,E1 -24922.482,E2 -24922.482} C_VEL
LIN {X 0,Y 134.225,Z 834.15,A -85,B 0,C 180,E1 -24926.995,E2 -24926.995} C_VEL
LIN {X 0,Y 134.212,Z 836.354,A -85,B 0,C 180,E1 -24929.997,E2 -24929.997} C_VEL
LIN {X 0,Y 133.981,Z 838.794,A -85,B 0,C 180,E1 -24934.684,E2 -24934.684} C_VEL
LIN {X 0,Y 133.958,Z 840.13,A -85,B 0,C 180,E1 -24939.052,E2 -24939.052} C_VEL
LIN {X 0,Y 135.227,Z 840.671,A -85,B 0,C 180,E1 -24945.058,E2 -24945.058} C_VEL
LIN {X 0,Y 135.566,Z 840.582,A -85,B 0,C 180,E1 -24946.034,E2 -24946.034} C_VEL
LIN {X 0,Y 135.98,Z 840.312,A -85,B 0,C 180,E1 -24948.52,E2 -24948.52} C_VEL
LIN {X 0,Y 135.572,Z 839.297,A -85,B 0,C 180,E1 -24952.684,E2 -24952.684} C_VEL
LIN {X 0,Y 135.685,Z 838.118,A -85,B 0,C 180,E1 -24955.998,E2 -24955.998} C_VEL
LIN {X 0,Y 136.826,Z 837.007,A -85,B 0,C 180,E1 -24958.386,E2 -24958.386} C_VEL
LIN {X 0,Y 137.505,Z 836.544,A -85,B 0,C 180,E1 -24959.136,E2 -24959.136} C_VEL
LIN {X 0,Y 143.698,Z 832.622,A -85,B 0,C 180,E1 -24964.221,E2 -24964.221} C_VEL
LIN {X 0,Y 149.275,Z 828.538,A -85,B 0,C 180,E1 -24967.734,E2 -24967.734} C_VEL
LIN {X 0,Y 155.509,Z 823.422,A -85,B 0,C 180,E1 -24970.939,E2 -24970.939} C_VEL
LIN {X 0,Y 163.46,Z 815.984,A -85,B 0,C 180,E1 -24974.317,E2 -24974.317} C_VEL
LIN {X 0,Y 170.815,Z 808.128,A -85,B 0,C 180,E1 -24976.908,E2 -24976.908} C_VEL
LIN {X 0,Y 178.602,Z 798.53,A -85,B 0,C 180,E1 -24979.239,E2 -24979.239} C_VEL
LIN {X 0,Y 186.168,Z 787.585,A -85,B 0,C 180,E1 -24981.129,E2 -24981.129} C_VEL
LIN {X 0,Y 192.534,Z 776.697,A -85,B 0,C 180,E1 -24982.55,E2 -24982.55} C_VEL
LIN {X 0,Y 198.403,Z 764.607,A -85,B 0,C 180,E1 -24983.69,E2 -24983.69} C_VEL
LIN {X 0,Y 202.891,Z 752.916,A -85,B 0,C 180,E1 -24984.512,E2 -24984.512} C_VEL
LIN {X 0,Y 207.045,Z 738.61,A -85,B 0,C 180,E1 -24985.228,E2 -24985.228} C_VEL
LIN {X 0,Y 209.601,Z 725.02,A -85,B 0,C 180,E1 -24985.765,E2 -24985.765} C_VEL
LIN {X 0,Y 209.098,Z 721.798,A -85,B 0,C 180,E1 -24987.577,E2 -24987.577} C_VEL
LIN {X 0,Y 208.694,Z 719.227,A -85,B 0,C 180,E1 -24989.47,E2 -24989.47} C_VEL
LIN {X 0,Y 208.474,Z 717.472,A -85,B 0,C 180,E1 -24992.073,E2 -24992.073} C_VEL
LIN {X 0,Y 208.585,Z 716.817,A -85,B 0,C 180,E1 -24994.022,E2 -24994.022} C_VEL
LIN {X 0,Y 209.34,Z 717.079,A -85,B 0,C 180,E1 -24997.28,E2 -24997.28} C_VEL
LIN {X 0,Y 210.329,Z 719.366,A -85,B 0,C 180,E1 -24999.918,E2 -24999.918} C_VEL
LIN {X 0,Y 207.464,Z 734.719,A -85,B 0,C 180,E1 -25000.592,E2 -25000.592} C_VEL
LIN {X 0,Y 203.804,Z 747.667,A -85,B 0,C 180,E1 -25001.415,E2 -25001.415} C_VEL
LIN {X 0,Y 199.189,Z 759.995,A -85,B 0,C 180,E1 -25002.519,E2 -25002.519} C_VEL
LIN {X 0,Y 193.425,Z 771.907,A -85,B 0,C 180,E1 -25003.915,E2 -25003.915} C_VEL
LIN {X 0,Y 187.146,Z 782.563,A -85,B 0,C 180,E1 -25005.592,E2 -25005.592} C_VEL
LIN {X 0,Y 179.787,Z 792.948,A -85,B 0,C 180,E1 -25007.747,E2 -25007.747} C_VEL
LIN {X 0,Y 172.901,Z 801.199,A -85,B 0,C 180,E1 -25010.052,E2 -25010.052} C_VEL
LIN {X 0,Y 165.806,Z 808.429,A -85,B 0,C 180,E1 -25012.694,E2 -25012.694} C_VEL
LIN {X 0,Y 157.999,Z 815.217,A -85,B 0,C 180,E1 -25016.174,E2 -25016.174} C_VEL
LIN {X 0,Y 150.854,Z 820.414,A -85,B 0,C 180,E1 -25020,E2 -25020} C_VEL
LIN {X 0,Y 144.448,Z 824.198,A -85,B 0,C 180,E1 -25024.185,E2 -25024.185} C_VEL
LIN {X 0,Y 139.013,Z 826.661,A -85,B 0,C 180,E1 -25028.723,E2 -25028.723} C_VEL
LIN {X 0,Y 135.901,Z 827.607,A -85,B 0,C 180,E1 -25031.938,E2 -25031.938} C_VEL
LIN {X 0,Y 132.172,Z 828.076,A -85,B 0,C 180,E1 -25036.853,E2 -25036.853} C_VEL
LIN {X 0,Y 129.157,Z 827.365,A -85,B 0,C 180,E1 -25042.389,E2 -25042.389} C_VEL
LIN {X 0,Y 127.268,Z 825.44,A -85,B 0,C 180,E1 -25047.934,E2 -25047.934} C_VEL
LIN {X 0,Y 126.435,Z 822.08,A -85,B 0,C 180,E1 -25053.769,E2 -25053.769} C_VEL
LIN {X 0,Y 126.566,Z 817.862,A -85,B 0,C 180,E1 -25058.983,E2 -25058.983} C_VEL
LIN {X 0,Y 127.333,Z 812.329,A -85,B 0,C 180,E1 -25064.155,E2 -25064.155} C_VEL
LIN {X 0,Y 128.599,Z 805.618,A -85,B 0,C 180,E1 -25069.024,E2 -25069.024} C_VEL
LIN {X 0,Y 130.529,Z 797.043,A -85,B 0,C 180,E1 -25073.865,E2 -25073.865} C_VEL
LIN {X 0,Y 132.981,Z 787.46,A -85,B 0,C 180,E1 -25078.1,E2 -25078.1} C_VEL
LIN {X 0,Y 135.589,Z 776.791,A -85,B 0,C 180,E1 -25081.782,E2 -25081.782} C_VEL
LIN {X 0,Y 138.128,Z 765.987,A -85,B 0,C 180,E1 -25084.698,E2 -25084.698} C_VEL
LIN {X 0,Y 140.59,Z 753.745,A -85,B 0,C 180,E1 -25087.271,E2 -25087.271} C_VEL
LIN {X 0,Y 142.786,Z 740.952,A -85,B 0,C 180,E1 -25089.258,E2 -25089.258} C_VEL
LIN {X 0,Y 144.419,Z 727.762,A -85,B 0,C 180,E1 -25090.748,E2 -25090.748} C_VEL
LIN {X 0,Y 145.926,Z 710.55,A -85,B 0,C 180,E1 -25091.937,E2 -25091.937} C_VEL
LIN {X 0,Y 148.669,Z 673.329,A -85,B 0,C 180,E1 -25094.132,E2 -25094.132} C_VEL
LIN {X 0,Y 139.582,Z 651.191,A -85,B 0,C 180,E1 -25097.536,E2 -25097.536} C_VEL
LIN {X 0,Y 130.795,Z 632.517,A -85,B 0,C 180,E1 -25101.117,E2 -25101.117} C_VEL
LIN {X 0,Y 129.645,Z 629.99,A -85,B 0,C 180,E1 -25101.626,E2 -25101.626} C_VEL
LIN {X 0,Y 129.549,Z 629.349,A -85,B 0,C 180,E1 -25101.816,E2 -25101.816} C_VEL
LIN {X 0,Y 130.091,Z 629.281,A -85,B 0,C 180,E1 -25110.003,E2 -25110.003} C_VEL
LIN {X 0,Y 129.533,Z 629.349,A -85,B 0,C 180,E1 -25119.371,E2 -25119.371} C_VEL
LIN {X 0,Y 129.395,Z 629.364,A -85,B 0,C 180,E1 -25122.551,E2 -25122.551} C_VEL
LIN {X 0,Y 129.157,Z 629.375,A -85,B 0,C 180,E1 -25129.059,E2 -25129.059} C_VEL
LIN {X 0,Y 129.111,Z 629.393,A -85,B 0,C 180,E1 -25132.401,E2 -25132.401} C_VEL
LIN {X 0,Y 129.039,Z 629.402,A -85,B 0,C 180,E1 -25139.376,E2 -25139.376} C_VEL
LIN {X 0,Y 128.964,Z 629.388,A -85,B 0,C 180,E1 -25145.171,E2 -25145.171} C_VEL
LIN {X 0,Y 128.938,Z 629.419,A -85,B 0,C 180,E1 -25150.854,E2 -25150.854} C_VEL
LIN {X 0,Y 128.926,Z 629.419,A -85,B 0,C 180,E1 -25155.13,E2 -25155.13} C_VEL
LIN {X 0,Y 128.947,Z 629.392,A -85,B 0,C 180,E1 -25159.738,E2 -25159.738} C_VEL
LIN {X 0,Y 128.986,Z 629.383,A -85,B 0,C 180,E1 -25164.821,E2 -25164.821} C_VEL
LIN {X 0,Y 129.022,Z 629.41,A -85,B 0,C 180,E1 -25170.644,E2 -25170.644} C_VEL
LIN {X 0,Y 129.034,Z 629.411,A -85,B 0,C 180,E1 -25174.169,E2 -25174.169} C_VEL
LIN {X 0,Y 129.114,Z 629.39,A -85,B 0,C 180,E1 -25177.73,E2 -25177.73} C_VEL
LIN {X 0,Y 129.189,Z 629.349,A -85,B 0,C 180,E1 -25184.217,E2 -25184.217} C_VEL
LIN {X 0,Y 129.383,Z 629.35,A -85,B 0,C 180,E1 -25187.905,E2 -25187.905} C_VEL
LIN {X 0,Y 129.481,Z 629.352,A -85,B 0,C 180,E1 -25190.629,E2 -25190.629} C_VEL
LIN {X 0,Y 130.096,Z 629.253,A -85,B 0,C 180,E1 -25200,E2 -25200} C_VEL
LIN {X 0,Y 129.48,Z 629.356,A -85,B 0,C 180,E1 -25209.372,E2 -25209.372} C_VEL
LIN {X 0,Y 129.307,Z 629.37,A -85,B 0,C 180,E1 -25212.557,E2 -25212.557} C_VEL
LIN {X 0,Y 129.122,Z 629.402,A -85,B 0,C 180,E1 -25219.062,E2 -25219.062} C_VEL
LIN {X 0,Y 129.114,Z 629.404,A -85,B 0,C 180,E1 -25222.398,E2 -25222.398} C_VEL
LIN {X 0,Y 129.043,Z 629.414,A -85,B 0,C 180,E1 -25229.372,E2 -25229.372} C_VEL
LIN {X 0,Y 128.967,Z 629.421,A -85,B 0,C 180,E1 -25235.168,E2 -25235.168} C_VEL
LIN {X 0,Y 129.008,Z 629.42,A -85,B 0,C 180,E1 -25241.863,E2 -25241.863} C_VEL
LIN {X 0,Y 130.277,Z 632.659,A -85,B 0,C 180,E1 -25242.534,E2 -25242.534} C_VEL
LIN {X 0,Y 136.916,Z 648.862,A -85,B 0,C 180,E1 -25245.49,E2 -25245.49} C_VEL
LIN {X 0,Y 144.26,Z 670.269,A -85,B 0,C 180,E1 -25248.639,E2 -25248.639} C_VEL
LIN {X 0,Y 145.848,Z 676.19,A -85,B 0,C 180,E1 -25249.372,E2 -25249.372} C_VEL
LIN {X 0,Y 147.543,Z 699.661,A -85,B 0,C 180,E1 -25251.37,E2 -25251.37} C_VEL
LIN {X 0,Y 144.472,Z 740.079,A -85,B 0,C 180,E1 -25253.851,E2 -25253.851} C_VEL
LIN {X 0,Y 142.899,Z 752.983,A -85,B 0,C 180,E1 -25255.125,E2 -25255.125} C_VEL
LIN {X 0,Y 140.923,Z 764.599,A -85,B 0,C 180,E1 -25256.727,E2 -25256.727} C_VEL
LIN {X 0,Y 138.346,Z 776.942,A -85,B 0,C 180,E1 -25259.042,E2 -25259.042} C_VEL
LIN {X 0,Y 135.851,Z 787.828,A -85,B 0,C 180,E1 -25261.734,E2 -25261.734} C_VEL
LIN {X 0,Y 133.288,Z 798.312,A -85,B 0,C 180,E1 -25265.047,E2 -25265.047} C_VEL
LIN {X 0,Y 131.016,Z 807.513,A -85,B 0,C 180,E1 -25268.768,E2 -25268.768} C_VEL
LIN {X 0,Y 129.009,Z 816.48,A -85,B 0,C 180,E1 -25273.378,E2 -25273.378} C_VEL
LIN {X 0,Y 127.763,Z 823.645,A -85,B 0,C 180,E1 -25278.092,E2 -25278.092} C_VEL
LIN {X 0,Y 127.285,Z 830.108,A -85,B 0,C 180,E1 -25283.657,E2 -25283.657} C_VEL
LIN {X 0,Y 127.166,Z 834.222,A -85,B 0,C 180,E1 -25288.413,E2 -25288.413} C_VEL
LIN {X 0,Y 127.186,Z 835.337,A -85,B 0,C 180,E1 -25289.997,E2 -25289.997} C_VEL
LIN {X 0,Y 126.947,Z 837.891,A -85,B 0,C 180,E1 -25294.782,E2 -25294.782} C_VEL
LIN {X 0,Y 126.962,Z 839.431,A -85,B 0,C 180,E1 -25299.556,E2 -25299.556} C_VEL
LIN {X 0,Y 128.37,Z 840.193,A -85,B 0,C 180,E1 -25305.883,E2 -25305.883} C_VEL
LIN {X 0,Y 131.413,Z 839.504,A -85,B 0,C 180,E1 -25311.981,E2 -25311.981} C_VEL
LIN {X 0,Y 136.064,Z 837.402,A -85,B 0,C 180,E1 -25317.698,E2 -25317.698} C_VEL
LIN {X 0,Y 137.505,Z 836.544,A -85,B 0,C 180,E1 -25319.136,E2 -25319.136} C_VEL
LIN {X 0,Y 139.286,Z 835.192,A -85,B 0,C 180,E1 -25321.409,E2 -25321.409} C_VEL
LIN {X 0,Y 141.062,Z 832.719,A -85,B 0,C 180,E1 -25325.283,E2 -25325.283} C_VEL
LIN {X 0,Y 143.529,Z 829.642,A -85,B 0,C 180,E1 -25328.927,E2 -25328.927} C_VEL
LIN {X 0,Y 146.267,Z 827.339,A -85,B 0,C 180,E1 -25330.767,E2 -25330.767} C_VEL
LIN {X 0,Y 152.549,Z 822.481,A -85,B 0,C 180,E1 -25333.709,E2 -25333.709} C_VEL
LIN {X 0,Y 161.001,Z 814.964,A -85,B 0,C 180,E1 -25336.98,E2 -25336.98} C_VEL
LIN {X 0,Y 170.087,Z 805.526,A -85,B 0,C 180,E1 -25339.851,E2 -25339.851} C_VEL
LIN {X 0,Y 176.965,Z 797.318,A -85,B 0,C 180,E1 -25341.656,E2 -25341.656} C_VEL
LIN {X 0,Y 184.81,Z 786.297,A -85,B 0,C 180,E1 -25343.446,E2 -25343.446} C_VEL
LIN {X 0,Y 191.426,Z 775.19,A -85,B 0,C 180,E1 -25344.77,E2 -25344.77} C_VEL
LIN {X 0,Y 197.441,Z 762.795,A -85,B 0,C 180,E1 -25345.848,E2 -25345.848} C_VEL
LIN {X 0,Y 202.05,Z 750.968,A -85,B 0,C 180,E1 -25346.591,E2 -25346.591} C_VEL
LIN {X 0,Y 206.102,Z 737.102,A -85,B 0,C 180,E1 -25347.225,E2 -25347.225} C_VEL
LIN {X 0,Y 207.69,Z 729.431,A -85,B 0,C 180,E1 -25347.535,E2 -25347.535} C_VEL
LIN {X 0,Y 207.34,Z 725.894,A -85,B 0,C 180,E1 -25350.01,E2 -25350.01} C_VEL
LIN {X 0,Y 207.202,Z 724.307,A -85,B 0,C 180,E1 -25352.549,E2 -25352.549} C_VEL
LIN {X 0,Y 207.307,Z 723.843,A -85,B 0,C 180,E1 -25353.85,E2 -25353.85} C_VEL
LIN {X 0,Y 208.014,Z 724.067,A -85,B 0,C 180,E1 -25357.127,E2 -25357.127} C_VEL
LIN {X 0,Y 208.326,Z 725.034,A -85,B 0,C 180,E1 -25358.217,E2 -25358.217} C_VEL
LIN {X 0,Y 205.144,Z 739.286,A -85,B 0,C 180,E1 -25358.874,E2 -25358.874} C_VEL
LIN {X 0,Y 201.253,Z 751.357,A -85,B 0,C 180,E1 -25359.694,E2 -25359.694} C_VEL
LIN {X 0,Y 195.824,Z 764.165,A -85,B 0,C 180,E1 -25360.883,E2 -25360.883} C_VEL
LIN {X 0,Y 189.862,Z 775.426,A -85,B 0,C 180,E1 -25362.258,E2 -25362.258} C_VEL
LIN {X 0,Y 183.846,Z 784.832,A -85,B 0,C 180,E1 -25363.763,E2 -25363.763} C_VEL
LIN {X 0,Y 177.027,Z 793.845,A -85,B 0,C 180,E1 -25365.633,E2 -25365.633} C_VEL
LIN {X 0,Y 169.353,Z 802.472,A -85,B 0,C 180,E1 -25368.024,E2 -25368.024} C_VEL
LIN {X 0,Y 161.931,Z 809.577,A -85,B 0,C 180,E1 -25370.633,E2 -25370.633} C_VEL
LIN {X 0,Y 154.327,Z 815.726,A -85,B 0,C 180,E1 -25373.784,E2 -25373.784} C_VEL
LIN {X 0,Y 147.28,Z 820.52,A -85,B 0,C 180,E1 -25377.265,E2 -25377.265} C_VEL
LIN {X 0,Y 140.585,Z 824.284,A -85,B 0,C 180,E1 -25381.247,E2 -25381.247} C_VEL
LIN {X 0,Y 134.261,Z 826.996,A -85,B 0,C 180,E1 -25386.009,E2 -25386.009} C_VEL
LIN {X 0,Y 128.972,Z 828.375,A -85,B 0,C 180,E1 -25391.246,E2 -25391.246} C_VEL
LIN {X 0,Y 124.815,Z 828.459,A -85,B 0,C 180,E1 -25396.832,E2 -25396.832} C_VEL
LIN {X 0,Y 121.831,Z 827.294,A -85,B 0,C 180,E1 -25402.644,E2 -25402.644} C_VEL
LIN {X 0,Y 119.996,Z 824.93,A -85,B 0,C 180,E1 -25408.543,E2 -25408.543} C_VEL
LIN {X 0,Y 119.303,Z 821.333,A -85,B 0,C 180,E1 -25414.446,E2 -25414.446} C_VEL
LIN {X 0,Y 119.594,Z 816.402,A -85,B 0,C 180,E1 -25420.272,E2 -25420.272} C_VEL
LIN {X 0,Y 120.523,Z 810.489,A -85,B 0,C 180,E1 -25425.599,E2 -25425.599} C_VEL
LIN {X 0,Y 121.982,Z 803.31,A -85,B 0,C 180,E1 -25430.677,E2 -25430.677} C_VEL
LIN {X 0,Y 124.108,Z 794.598,A -85,B 0,C 180,E1 -25435.513,E2 -25435.513} C_VEL
LIN {X 0,Y 126.485,Z 785.525,A -85,B 0,C 180,E1 -25439.455,E2 -25439.455} C_VEL
LIN {X 0,Y 129.116,Z 775.139,A -85,B 0,C 180,E1 -25443.039,E2 -25443.039} C_VEL
LIN {X 0,Y 131.985,Z 763.13,A -85,B 0,C 180,E1 -25446.235,E2 -25446.235} C_VEL
LIN {X 0,Y 134.551,Z 750.278,A -85,B 0,C 180,E1 -25448.833,E2 -25448.833} C_VEL
LIN {X 0,Y 136.589,Z 737.968,A -85,B 0,C 180,E1 -25450.66,E2 -25450.66} C_VEL
LIN {X 0,Y 138.232,Z 723.725,A -85,B 0,C 180,E1 -25452.146,E2 -25452.146} C_VEL
LIN {X 0,Y 142.127,Z 674.966,A -85,B 0,C 180,E1 -25455.195,E2 -25455.195} C_VEL
LIN {X 0,Y 133.185,Z 653.03,A -85,B 0,C 180,E1 -25458.836,E2 -25458.836} C_VEL
LIN {X 0,Y 125.412,Z 636.519,A -85,B 0,C 180,E1 -25462.178,E2 -25462.178} C_VEL
LIN {X 0,Y 122.692,Z 631.299,A -85,B 0,C 180,E1 -25463.425,E2 -25463.425} C_VEL
LIN {X 0,Y 122.468,Z 630.232,A -85,B 0,C 180,E1 -25463.62,E2 -25463.62} C_VEL
LIN {X 0,Y 123.045,Z 630.159,A -85,B 0,C 180,E1 -25470.004,E2 -25470.004} C_VEL
LIN {X 0,Y 122.459,Z 630.228,A -85,B 0,C 180,E1 -25476.595,E2 -25476.595} C_VEL
LIN {X 0,Y 122.459,Z 630.23,A -85,B 0,C 180,E1 -25479.918,E2 -25479.918} C_VEL
LIN {X 0,Y 122.265,Z 630.255,A -85,B 0,C 180,E1 -25483.296,E2 -25483.296} C_VEL
LIN {X 0,Y 122.048,Z 630.26,A -85,B 0,C 180,E1 -25490.216,E2 -25490.216} C_VEL
LIN {X 0,Y 121.987,Z 630.287,A -85,B 0,C 180,E1 -25493.788,E2 -25493.788} C_VEL
LIN {X 0,Y 121.943,Z 630.282,A -85,B 0,C 180,E1 -25500.175,E2 -25500.175} C_VEL
LIN {X 0,Y 121.888,Z 630.276,A -85,B 0,C 180,E1 -25506.174,E2 -25506.174} C_VEL
LIN {X 0,Y 121.877,Z 630.301,A -85,B 0,C 180,E1 -25511.441,E2 -25511.441} C_VEL
LIN {X 0,Y 121.877,Z 630.279,A -85,B 0,C 180,E1 -25518.564,E2 -25518.564} C_VEL
LIN {X 0,Y 121.938,Z 630.258,A -85,B 0,C 180,E1 -25524.806,E2 -25524.806} C_VEL
LIN {X 0,Y 121.935,Z 630.29,A -85,B 0,C 180,E1 -25529.839,E2 -25529.839} C_VEL
LIN {X 0,Y 121.989,Z 630.284,A -85,B 0,C 180,E1 -25536.217,E2 -25536.217} C_VEL
LIN {X 0,Y 122.038,Z 630.259,A -85,B 0,C 180,E1 -25539.786,E2 -25539.786} C_VEL
LIN {X 0,Y 122.244,Z 630.229,A -85,B 0,C 180,E1 -25546.705,E2 -25546.705} C_VEL
LIN {X 0,Y 122.414,Z 630.228,A -85,B 0,C 180,E1 -25550.083,E2 -25550.083} C_VEL
LIN {X 0,Y 122.605,Z 630.205,A -85,B 0,C 180,E1 -25556.714,E2 -25556.714} C_VEL
LIN {X 0,Y 123.049,Z 630.13,A -85,B 0,C 180,E1 -25560,E2 -25560} C_VEL
LIN {X 0,Y 122.432,Z 630.228,A -85,B 0,C 180,E1 -25566.593,E2 -25566.593} C_VEL
LIN {X 0,Y 122.406,Z 630.238,A -85,B 0,C 180,E1 -25569.919,E2 -25569.919} C_VEL
LIN {X 0,Y 122.197,Z 630.253,A -85,B 0,C 180,E1 -25573.301,E2 -25573.301} C_VEL
LIN {X 0,Y 122.028,Z 630.288,A -85,B 0,C 180,E1 -25580.217,E2 -25580.217} C_VEL
LIN {X 0,Y 121.989,Z 630.286,A -85,B 0,C 180,E1 -25583.784,E2 -25583.784} C_VEL
LIN {X 0,Y 121.947,Z 630.299,A -85,B 0,C 180,E1 -25590.171,E2 -25590.171} C_VEL
LIN {X 0,Y 121.891,Z 630.302,A -85,B 0,C 180,E1 -25596.17,E2 -25596.17} C_VEL
LIN {X 0,Y 121.951,Z 630.437,A -85,B 0,C 180,E1 -25600.037,E2 -25600.037} C_VEL
LIN {X 0,Y 123.074,Z 633.351,A -85,B 0,C 180,E1 -25600.64,E2 -25600.64} C_VEL
LIN {X 0,Y 125.389,Z 637.74,A -85,B 0,C 180,E1 -25601.69,E2 -25601.69} C_VEL
LIN {X 0,Y 132.034,Z 654.569,A -85,B 0,C 180,E1 -25604.829,E2 -25604.829} C_VEL
LIN {X 0,Y 138.826,Z 675.172,A -85,B 0,C 180,E1 -25607.967,E2 -25607.967} C_VEL
LIN {X 0,Y 139.538,Z 678.784,A -85,B 0,C 180,E1 -25608.386,E2 -25608.386} C_VEL
LIN {X 0,Y 141.03,Z 699.66,A -85,B 0,C 180,E1 -25610.247,E2 -25610.247} C_VEL
LIN {X 0,Y 137.825,Z 739.954,A -85,B 0,C 180,E1 -25612.844,E2 -25612.844} C_VEL
LIN {X 0,Y 136.132,Z 753.436,A -85,B 0,C 180,E1 -25614.262,E2 -25614.262} C_VEL
LIN {X 0,Y 133.885,Z 765.737,A -85,B 0,C 180,E1 -25616.097,E2 -25616.097} C_VEL
LIN {X 0,Y 131.222,Z 777.691,A -85,B 0,C 180,E1 -25618.518,E2 -25618.518} C_VEL
LIN {X 0,Y 128.61,Z 788.677,A -85,B 0,C 180,E1 -25621.437,E2 -25621.437} C_VEL
LIN {X 0,Y 125.835,Z 799.625,A -85,B 0,C 180,E1 -25625.232,E2 -25625.232} C_VEL
LIN {X 0,Y 123.578,Z 808.532,A -85,B 0,C 180,E1 -25629.176,E2 -25629.176} C_VEL
LIN {X 0,Y 121.945,Z 815.899,A -85,B 0,C 180,E1 -25633.248,E2 -25633.248} C_VEL
LIN {X 0,Y 120.683,Z 823.097,A -85,B 0,C 180,E1 -25638.236,E2 -25638.236} C_VEL
LIN {X 0,Y 120.25,Z 828.981,A -85,B 0,C 180,E1 -25643.501,E2 -25643.501} C_VEL
LIN {X 0,Y 120.163,Z 833.083,A -85,B 0,C 180,E1 -25648.321,E2 -25648.321} C_VEL
LIN {X 0,Y 120.182,Z 834.254,A -85,B 0,C 180,E1 -25649.996,E2 -25649.996} C_VEL
LIN {X 0,Y 119.919,Z 836.887,A -85,B 0,C 180,E1 -25654.922,E2 -25654.922} C_VEL
LIN {X 0,Y 119.986,Z 838.66,A -85,B 0,C 180,E1 -25660.117,E2 -25660.117} C_VEL
LIN {X 0,Y 121.527,Z 839.672,A -85,B 0,C 180,E1 -25666.803,E2 -25666.803} C_VEL
LIN {X 0,Y 122.903,Z 839.637,A -85,B 0,C 180,E1 -25670.062,E2 -25670.062} C_VEL
LIN {X 0,Y 127.108,Z 838.469,A -85,B 0,C 180,E1 -25676.249,E2 -25676.249} C_VEL
LIN {X 0,Y 132.772,Z 835.88,A -85,B 0,C 180,E1 -25681.956,E2 -25681.956} C_VEL
LIN {X 0,Y 139.773,Z 831.801,A -85,B 0,C 180,E1 -25687.108,E2 -25687.108} C_VEL
LIN {X 0,Y 146.267,Z 827.339,A -85,B 0,C 180,E1 -25690.767,E2 -25690.767} C_VEL
LIN {X 0,Y 149.176,Z 824.927,A -85,B 0,C 180,E1 -25692.519,E2 -25692.519} C_VEL
LIN {X 0,Y 155.75,Z 817.286,A -85,B 0,C 180,E1 -25698.068,E2 -25698.068} C_VEL
LIN {X 0,Y 158.695,Z 814.273,A -85,B 0,C 180,E1 -25699.564,E2 -25699.564} C_VEL
LIN {X 0,Y 159.873,Z 813.163,A -85,B 0,C 180,E1 -25699.968,E2 -25699.968} C_VEL
LIN {X 0,Y 168.495,Z 804.529,A -85,B 0,C 180,E1 -25702.415,E2 -25702.415} C_VEL
LIN {X 0,Y 177.117,Z 794.302,A -85,B 0,C 180,E1 -25704.429,E2 -25704.429} C_VEL
LIN {X 0,Y 185.281,Z 782.815,A -85,B 0,C 180,E1 -25706.068,E2 -25706.068} C_VEL
LIN {X 0,Y 192.166,Z 771.015,A -85,B 0,C 180,E1 -25707.259,E2 -25707.259} C_VEL
LIN {X 0,Y 197.595,Z 759.584,A -85,B 0,C 180,E1 -25708.118,E2 -25708.118} C_VEL
LIN {X 0,Y 202.56,Z 746.166,A -85,B 0,C 180,E1 -25708.816,E2 -25708.816} C_VEL
LIN {X 0,Y 205.793,Z 734.142,A -85,B 0,C 180,E1 -25709.354,E2 -25709.354} C_VEL
LIN {X 0,Y 205.826,Z 732.364,A -85,B 0,C 180,E1 -25710.798,E2 -25710.798} C_VEL
LIN {X 0,Y 205.896,Z 730.855,A -85,B 0,C 180,E1 -25713.657,E2 -25713.657} C_VEL
LIN {X 0,Y 206.351,Z 730.95,A -85,B 0,C 180,E1 -25716.491,E2 -25716.491} C_VEL
LIN {X 0,Y 203.093,Z 743.226,A -85,B 0,C 180,E1 -25717.116,E2 -25717.116} C_VEL
LIN {X 0,Y 198.512,Z 755.973,A -85,B 0,C 180,E1 -25718.003,E2 -25718.003} C_VEL
LIN {X 0,Y 192.743,Z 768.179,A -85,B 0,C 180,E1 -25719.175,E2 -25719.175} C_VEL
LIN {X 0,Y 186.291,Z 779.178,A -85,B 0,C 180,E1 -25720.579,E2 -25720.579} C_VEL
LIN {X 0,Y 179.139,Z 789.203,A -85,B 0,C 180,E1 -25722.29,E2 -25722.29} C_VEL
LIN {X 0,Y 172.47,Z 797.189,A -85,B 0,C 180,E1 -25724.034,E2 -25724.034} C_VEL
LIN {X 0,Y 164.502,Z 805.299,A -85,B 0,C 180,E1 -25726.408,E2 -25726.408} C_VEL
LIN {X 0,Y 157.67,Z 811.211,A -85,B 0,C 180,E1 -25728.689,E2 -25728.689} C_VEL
LIN {X 0,Y 148.975,Z 817.662,A -85,B 0,C 180,E1 -25732.151,E2 -25732.151} C_VEL
LIN {X 0,Y 140.882,Z 822.525,A -85,B 0,C 180,E1 -25736.076,E2 -25736.076} C_VEL
LIN {X 0,Y 133.528,Z 825.97,A -85,B 0,C 180,E1 -25740.467,E2 -25740.467} C_VEL
LIN {X 0,Y 127.066,Z 828.154,A -85,B 0,C 180,E1 -25745.431,E2 -25745.431} C_VEL
LIN {X 0,Y 121.668,Z 829.061,A -85,B 0,C 180,E1 -25750.914,E2 -25750.914} C_VEL
LIN {X 0,Y 117.069,Z 828.555,A -85,B 0,C 180,E1 -25757.467,E2 -25757.467} C_VEL
LIN {X 0,Y 114.471,Z 827.067,A -85,B 0,C 180,E1 -25762.948,E2 -25762.948} C_VEL
LIN {X 0,Y 112.624,Z 823.846,A -85,B 0,C 180,E1 -25769.948,E2 -25769.948} C_VEL
LIN {X 0,Y 112.257,Z 819.043,A -85,B 0,C 180,E1 -25776.97,E2 -25776.97} C_VEL
LIN {X 0,Y 112.923,Z 813.172,A -85,B 0,C 180,E1 -25783.204,E2 -25783.204} C_VEL
LIN {X 0,Y 114.239,Z 806.199,A -85,B 0,C 180,E1 -25788.904,E2 -25788.904} C_VEL
LIN {X 0,Y 116.129,Z 798.123,A -85,B 0,C 180,E1 -25794.037,E2 -25794.037} C_VEL
LIN {X 0,Y 118.655,Z 788.587,A -85,B 0,C 180,E1 -25798.8,E2 -25798.8} C_VEL
LIN {X 0,Y 121.502,Z 778.106,A -85,B 0,C 180,E1 -25802.866,E2 -25802.866} C_VEL
LIN {X 0,Y 124.595,Z 765.706,A -85,B 0,C 180,E1 -25806.555,E2 -25806.555} C_VEL
LIN {X 0,Y 127.13,Z 754.078,A -85,B 0,C 180,E1 -25809.18,E2 -25809.18} C_VEL
LIN {X 0,Y 129.617,Z 740.355,A -85,B 0,C 180,E1 -25811.463,E2 -25811.463} C_VEL
LIN {X 0,Y 131.381,Z 726.818,A -85,B 0,C 180,E1 -25813.03,E2 -25813.03} C_VEL
LIN {X 0,Y 133.255,Z 705.53,A -85,B 0,C 180,E1 -25814.536,E2 -25814.536} C_VEL
LIN {X 0,Y 135.649,Z 676.963,A -85,B 0,C 180,E1 -25816.337,E2 -25816.337} C_VEL
LIN {X 0,Y 128.197,Z 658.172,A -85,B 0,C 180,E1 -25819.566,E2 -25819.566} C_VEL
LIN {X 0,Y 120.069,Z 640.513,A -85,B 0,C 180,E1 -25823.334,E2 -25823.334} C_VEL
LIN {X 0,Y 116.607,Z 634.133,A -85,B 0,C 180,E1 -25825.034,E2 -25825.034} C_VEL
LIN {X 0,Y 115.548,Z 631.402,A -85,B 0,C 180,E1 -25825.643,E2 -25825.643} C_VEL
LIN {X 0,Y 115.499,Z 631.099,A -85,B 0,C 180,E1 -25825.86,E2 -25825.86} C_VEL
LIN {X 0,Y 115.997,Z 631.037,A -85,B 0,C 180,E1 -25830.004,E2 -25830.004} C_VEL
LIN {X 0,Y 115.4,Z 631.107,A -85,B 0,C 180,E1 -25837,E2 -25837} C_VEL
LIN {X 0,Y 115.395,Z 631.108,A -85,B 0,C 180,E1 -25840.532,E2 -25840.532} C_VEL
LIN {X 0,Y 115.148,Z 631.141,A -85,B 0,C 180,E1 -25844.135,E2 -25844.135} C_VEL
LIN {X 0,Y 114.982,Z 631.146,A -85,B 0,C 180,E1 -25851.518,E2 -25851.518} C_VEL
LIN {X 0,Y 114.877,Z 631.176,A -85,B 0,C 180,E1 -25855.36,E2 -25855.36} C_VEL
LIN {X 0,Y 114.866,Z 631.157,A -85,B 0,C 180,E1 -25861.066,E2 -25861.066} C_VEL
LIN {X 0,Y 114.784,Z 631.17,A -85,B 0,C 180,E1 -25867.759,E2 -25867.759} C_VEL
LIN {X 0,Y 114.792,Z 631.183,A -85,B 0,C 180,E1 -25872.72,E2 -25872.72} C_VEL
LIN {X 0,Y 114.799,Z 631.166,A -85,B 0,C 180,E1 -25877.669,E2 -25877.669} C_VEL
LIN {X 0,Y 114.802,Z 631.133,A -85,B 0,C 180,E1 -25882.74,E2 -25882.74} C_VEL
LIN {X 0,Y 114.868,Z 631.167,A -85,B 0,C 180,E1 -25888.94,E2 -25888.94} C_VEL
LIN {X 0,Y 114.953,Z 631.159,A -85,B 0,C 180,E1 -25896.51,E2 -25896.51} C_VEL
LIN {X 0,Y 115.006,Z 631.115,A -85,B 0,C 180,E1 -25902.209,E2 -25902.209} C_VEL
LIN {X 0,Y 115.262,Z 631.103,A -85,B 0,C 180,E1 -25907.328,E2 -25907.328} C_VEL
LIN {X 0,Y 115.373,Z 631.112,A -85,B 0,C 180,E1 -25913.003,E2 -25913.003} C_VEL
LIN {X 0,Y 116.001,Z 631.007,A -85,B 0,C 180,E1 -25920,E2 -25920} C_VEL
LIN {X 0,Y 115.371,Z 631.11,A -85,B 0,C 180,E1 -25926.998,E2 -25926.998} C_VEL
LIN {X 0,Y 115.213,Z 631.125,A -85,B 0,C 180,E1 -25932.563,E2 -25932.563} C_VEL
LIN {X 0,Y 114.992,Z 631.155,A -85,B 0,C 180,E1 -25937.794,E2 -25937.794} C_VEL
LIN {X 0,Y 114.952,Z 631.164,A -85,B 0,C 180,E1 -25943.489,E2 -25943.489} C_VEL
LIN {X 0,Y 114.869,Z 631.176,A -85,B 0,C 180,E1 -25951.061,E2 -25951.061} C_VEL
LIN {X 0,Y 114.821,Z 631.194,A -85,B 0,C 180,E1 -25957.88,E2 -25957.88} C_VEL
LIN {X 0,Y 115.783,Z 633.987,A -85,B 0,C 180,E1 -25958.476,E2 -25958.476} C_VEL
LIN {X 0,Y 117.373,Z 636.571,A -85,B 0,C 180,E1 -25959.232,E2 -25959.232} C_VEL
LIN {X 0,Y 120.177,Z 642.181,A -85,B 0,C 180,E1 -25960.632,E2 -25960.632} C_VEL
LIN {X 0,Y 126.523,Z 658.602,A -85,B 0,C 180,E1 -25963.837,E2 -25963.837} C_VEL
LIN {X 0,Y 133.048,Z 678.832,A -85,B 0,C 180,E1 -25967.062,E2 -25967.062} C_VEL
LIN {X 0,Y 134.454,Z 701.063,A -85,B 0,C 180,E1 -25969.138,E2 -25969.138} C_VEL
LIN {X 0,Y 131.243,Z 739.648,A -85,B 0,C 180,E1 -25971.741,E2 -25971.741} C_VEL
LIN {X 0,Y 129.374,Z 753.753,A -85,B 0,C 180,E1 -25973.301,E2 -25973.301} C_VEL
LIN {X 0,Y 126.844,Z 766.756,A -85,B 0,C 180,E1 -25975.391,E2 -25975.391} C_VEL
LIN {X 0,Y 123.973,Z 779.189,A -85,B 0,C 180,E1 -25978.122,E2 -25978.122} C_VEL
LIN {X 0,Y 121.093,Z 790.452,A -85,B 0,C 180,E1 -25981.439,E2 -25981.439} C_VEL
LIN {X 0,Y 118.379,Z 800.928,A -85,B 0,C 180,E1 -25985.44,E2 -25985.44} C_VEL
LIN {X 0,Y 116.191,Z 809.513,A -85,B 0,C 180,E1 -25989.643,E2 -25989.643} C_VEL
LIN {X 0,Y 114.322,Z 817.821,A -85,B 0,C 180,E1 -25994.851,E2 -25994.851} C_VEL
LIN {X 0,Y 113.485,Z 823.489,A -85,B 0,C 180,E1 -25999.289,E2 -25999.289} C_VEL
LIN {X 0,Y 113.205,Z 829.224,A -85,B 0,C 180,E1 -26004.954,E2 -26004.954} C_VEL
LIN {X 0,Y 113.175,Z 833.079,A -85,B 0,C 180,E1 -26009.996,E2 -26009.996} C_VEL
LIN {X 0,Y 112.909,Z 835.896,A -85,B 0,C 180,E1 -26015.174,E2 -26015.174} C_VEL
LIN {X 0,Y 113.003,Z 837.873,A -85,B 0,C 180,E1 -26020.749,E2 -26020.749} C_VEL
LIN {X 0,Y 114.727,Z 839.082,A -85,B 0,C 180,E1 -26027.832,E2 -26027.832} C_VEL
LIN {X 0,Y 118.337,Z 838.902,A -85,B 0,C 180,E1 -26034.561,E2 -26034.561} C_VEL
LIN {X 0,Y 123.629,Z 837.321,A -85,B 0,C 180,E1 -26040.768,E2 -26040.768} C_VEL
LIN {X 0,Y 130.334,Z 834.254,A -85,B 0,C 180,E1 -26046.377,E2 -26046.377} C_VEL
LIN {X 0,Y 138.366,Z 829.708,A -85,B 0,C 180,E1 -26051.319,E2 -26051.319} C_VEL
LIN {X 0,Y 145.168,Z 825.171,A -85,B 0,C 180,E1 -26054.582,E2 -26054.582} C_VEL
LIN {X 0,Y 153.777,Z 818.522,A -85,B 0,C 180,E1 -26057.954,E2 -26057.954} C_VEL
LIN {X 0,Y 159.873,Z 813.163,A -85,B 0,C 180,E1 -26059.968,E2 -26059.968} C_VEL
LIN {X 0,Y 163.207,Z 809.845,A -85,B 0,C 180,E1 -26061.24,E2 -26061.24} C_VEL
LIN {X 0,Y 167.719,Z 804.373,A -85,B 0,C 180,E1 -26063.642,E2 -26063.642} C_VEL
LIN {X 0,Y 172.22,Z 798.409,A -85,B 0,C 180,E1 -26065.811,E2 -26065.811} C_VEL
LIN {X 0,Y 175.416,Z 794.335,A -85,B 0,C 180,E1 -26066.721,E2 -26066.721} C_VEL
LIN {X 0,Y 183.844,Z 782.947,A -85,B 0,C 180,E1 -26068.269,E2 -26068.269} C_VEL
LIN {X 0,Y 190.923,Z 771.229,A -85,B 0,C 180,E1 -26069.362,E2 -26069.362} C_VEL
LIN {X 0,Y 197.351,Z 758.131,A -85,B 0,C 180,E1 -26070.27,E2 -26070.27} C_VEL
LIN {X 0,Y 202.512,Z 744.22,A -85,B 0,C 180,E1 -26070.906,E2 -26070.906} C_VEL
LIN {X 0,Y 204.008,Z 739.119,A -85,B 0,C 180,E1 -26071.164,E2 -26071.164} C_VEL
LIN {X 0,Y 204.125,Z 737.795,A -85,B 0,C 180,E1 -26073.525,E2 -26073.525} C_VEL
LIN {X 0,Y 204.279,Z 737.688,A -85,B 0,C 180,E1 -26074.776,E2 -26074.776} C_VEL
LIN {X 0,Y 199.919,Z 751.07,A -85,B 0,C 180,E1 -26075.565,E2 -26075.565} C_VEL
LIN {X 0,Y 194.992,Z 762.39,A -85,B 0,C 180,E1 -26076.451,E2 -26076.451} C_VEL
LIN {X 0,Y 187.997,Z 775.096,A -85,B 0,C 180,E1 -26077.785,E2 -26077.785} C_VEL
LIN {X 0,Y 181.49,Z 784.782,A -85,B 0,C 180,E1 -26079.132,E2 -26079.132} C_VEL
LIN {X 0,Y 173.139,Z 795.022,A -85,B 0,C 180,E1 -26081.05,E2 -26081.05} C_VEL
LIN {X 0,Y 164.866,Z 803.484,A -85,B 0,C 180,E1 -26083.211,E2 -26083.211} C_VEL
LIN {X 0,Y 156.517,Z 810.716,A -85,B 0,C 180,E1 -26085.702,E2 -26085.702} C_VEL
LIN {X 0,Y 149.536,Z 815.841,A -85,B 0,C 180,E1 -26088.091,E2 -26088.091} C_VEL
LIN {X 0,Y 141.359,Z 820.882,A -85,B 0,C 180,E1 -26091.422,E2 -26091.422} C_VEL
LIN {X 0,Y 134.03,Z 824.594,A -85,B 0,C 180,E1 -26095.017,E2 -26095.017} C_VEL
LIN {X 0,Y 125.88,Z 827.682,A -85,B 0,C 180,E1 -26100,E2 -26100} C_VEL
LIN {X 0,Y 119.881,Z 829.132,A -85,B 0,C 180,E1 -26104.762,E2 -26104.762} C_VEL
LIN {X 0,Y 114.296,Z 829.548,A -85,B 0,C 180,E1 -26110.63,E2 -26110.63} C_VEL
LIN {X 0,Y 110.091,Z 828.729,A -85,B 0,C 180,E1 -26116.765,E2 -26116.765} C_VEL
LIN {X 0,Y 107.115,Z 826.684,A -85,B 0,C 180,E1 -26123.294,E2 -26123.294} C_VEL
LIN {X 0,Y 105.511,Z 823.37,A -85,B 0,C 180,E1 -26130.021,E2 -26130.021} C_VEL
LIN {X 0,Y 105.173,Z 818.612,A -85,B 0,C 180,E1 -26136.97,E2 -26136.97} C_VEL
LIN {X 0,Y 105.796,Z 813.112,A -85,B 0,C 180,E1 -26143.059,E2 -26143.059} C_VEL
LIN {X 0,Y 107.125,Z 806.213,A -85,B 0,C 180,E1 -26149.006,E2 -26149.006} C_VEL
LIN {X 0,Y 109.135,Z 797.844,A -85,B 0,C 180,E1 -26154.584,E2 -26154.584} C_VEL
LIN {X 0,Y 111.543,Z 789.027,A -85,B 0,C 180,E1 -26159.219,E2 -26159.219} C_VEL
LIN {X 0,Y 114.511,Z 778.453,A -85,B 0,C 180,E1 -26163.556,E2 -26163.556} C_VEL
LIN {X 0,Y 117.328,Z 767.399,A -85,B 0,C 180,E1 -26167.068,E2 -26167.068} C_VEL
LIN {X 0,Y 120.152,Z 755.463,A -85,B 0,C 180,E1 -26169.973,E2 -26169.973} C_VEL
LIN {X 0,Y 122.706,Z 742.078,A -85,B 0,C 180,E1 -26172.368,E2 -26172.368} C_VEL
LIN {X 0,Y 124.586,Z 728.986,A -85,B 0,C 180,E1 -26174.044,E2 -26174.044} C_VEL
LIN {X 0,Y 126.279,Z 711.705,A -85,B 0,C 180,E1 -26175.405,E2 -26175.405} C_VEL
LIN {X 0,Y 129.132,Z 678.306,A -85,B 0,C 180,E1 -26177.629,E2 -26177.629} C_VEL
LIN {X 0,Y 121.089,Z 658.41,A -85,B 0,C 180,E1 -26181.366,E2 -26181.366} C_VEL
LIN {X 0,Y 114.376,Z 643.737,A -85,B 0,C 180,E1 -26184.771,E2 -26184.771} C_VEL
LIN {X 0,Y 108.806,Z 632.944,A -85,B 0,C 180,E1 -26187.806,E2 -26187.806} C_VEL
LIN {X 0,Y 108.646,Z 631.952,A -85,B 0,C 180,E1 -26188.151,E2 -26188.151} C_VEL
LIN {X 0,Y 108.948,Z 631.915,A -85,B 0,C 180,E1 -26190.004,E2 -26190.004} C_VEL
LIN {X 0,Y 108.342,Z 631.987,A -85,B 0,C 180,E1 -26197.458,E2 -26197.458} C_VEL
LIN {X 0,Y 108.205,Z 632.006,A -85,B 0,C 180,E1 -26203.029,E2 -26203.029} C_VEL
LIN {X 0,Y 107.908,Z 632.02,A -85,B 0,C 180,E1 -26209.009,E2 -26209.009} C_VEL
LIN {X 0,Y 107.862,Z 632.046,A -85,B 0,C 180,E1 -26214.19,E2 -26214.19} C_VEL
LIN {X 0,Y 107.788,Z 632.027,A -85,B 0,C 180,E1 -26222.046,E2 -26222.046} C_VEL
LIN {X 0,Y 107.693,Z 632.058,A -85,B 0,C 180,E1 -26228.454,E2 -26228.454} C_VEL
LIN {X 0,Y 107.682,Z 632.061,A -85,B 0,C 180,E1 -26235.889,E2 -26235.889} C_VEL
LIN {X 0,Y 107.698,Z 632.018,A -85,B 0,C 180,E1 -26241.549,E2 -26241.549} C_VEL
LIN {X 0,Y 107.806,Z 632.044,A -85,B 0,C 180,E1 -26248.566,E2 -26248.566} C_VEL
LIN {X 0,Y 107.916,Z 632.033,A -85,B 0,C 180,E1 -26257,E2 -26257} C_VEL
LIN {X 0,Y 108.032,Z 631.982,A -85,B 0,C 180,E1 -26264.917,E2 -26264.917} C_VEL
LIN {X 0,Y 108.263,Z 631.983,A -85,B 0,C 180,E1 -26268.77,E2 -26268.77} C_VEL
LIN {X 0,Y 108.453,Z 631.968,A -85,B 0,C 180,E1 -26276.285,E2 -26276.285} C_VEL
LIN {X 0,Y 108.926,Z 631.887,A -85,B 0,C 180,E1 -26280.001,E2 -26280.001} C_VEL
LIN {X 0,Y 108.308,Z 631.991,A -85,B 0,C 180,E1 -26287.457,E2 -26287.457} C_VEL
LIN {X 0,Y 108.147,Z 632.004,A -85,B 0,C 180,E1 -26292.877,E2 -26292.877} C_VEL
LIN {X 0,Y 107.891,Z 632.045,A -85,B 0,C 180,E1 -26299.009,E2 -26299.009} C_VEL
LIN {X 0,Y 107.864,Z 632.042,A -85,B 0,C 180,E1 -26304.182,E2 -26304.182} C_VEL
LIN {X 0,Y 107.791,Z 632.053,A -85,B 0,C 180,E1 -26312.041,E2 -26312.041} C_VEL
LIN {X 0,Y 107.727,Z 632.067,A -85,B 0,C 180,E1 -26315.415,E2 -26315.415} C_VEL
LIN {X 0,Y 108.717,Z 634.889,A -85,B 0,C 180,E1 -26316.145,E2 -26316.145} C_VEL
LIN {X 0,Y 110.115,Z 637.087,A -85,B 0,C 180,E1 -26316.881,E2 -26316.881} C_VEL
LIN {X 0,Y 114.425,Z 645.092,A -85,B 0,C 180,E1 -26319.16,E2 -26319.16} C_VEL
LIN {X 0,Y 120.533,Z 661.246,A -85,B 0,C 180,E1 -26322.533,E2 -26322.533} C_VEL
LIN {X 0,Y 126.782,Z 680.735,A -85,B 0,C 180,E1 -26325.822,E2 -26325.822} C_VEL
LIN {X 0,Y 128.053,Z 700.724,A -85,B 0,C 180,E1 -26327.811,E2 -26327.811} C_VEL
LIN {X 0,Y 124.716,Z 739.266,A -85,B 0,C 180,E1 -26330.522,E2 -26330.522} C_VEL
LIN {X 0,Y 122.861,Z 752.587,A -85,B 0,C 180,E1 -26332.049,E2 -26332.049} C_VEL
LIN {X 0,Y 120.692,Z 763.889,A -85,B 0,C 180,E1 -26333.868,E2 -26333.868} C_VEL
LIN {X 0,Y 117.945,Z 775.542,A -85,B 0,C 180,E1 -26336.396,E2 -26336.396} C_VEL
LIN {X 0,Y 114.909,Z 787.374,A -85,B 0,C 180,E1 -26339.819,E2 -26339.819} C_VEL
LIN {X 0,Y 111.974,Z 798.145,A -85,B 0,C 180,E1 -26343.933,E2 -26343.933} C_VEL
LIN {X 0,Y 109.578,Z 807.122,A -85,B 0,C 180,E1 -26348.355,E2 -26348.355} C_VEL
LIN {X 0,Y 107.549,Z 815.892,A -85,B 0,C 180,E1 -26353.871,E2 -26353.871} C_VEL
LIN {X 0,Y 106.414,Z 822.836,A -85,B 0,C 180,E1 -26359.532,E2 -26359.532} C_VEL
LIN {X 0,Y 106.194,Z 827.875,A -85,B 0,C 180,E1 -26364.691,E2 -26364.691} C_VEL
LIN {X 0,Y 106.167,Z 831.899,A -85,B 0,C 180,E1 -26369.996,E2 -26369.996} C_VEL
LIN {X 0,Y 105.893,Z 834.803,A -85,B 0,C 180,E1 -26375.412,E2 -26375.412} C_VEL
LIN {X 0,Y 106.075,Z 836.994,A -85,B 0,C 180,E1 -26381.461,E2 -26381.461} C_VEL
LIN {X 0,Y 107.976,Z 838.488,A -85,B 0,C 180,E1 -26388.988,E2 -26388.988} C_VEL
LIN {X 0,Y 111.909,Z 838.533,A -85,B 0,C 180,E1 -26396.074,E2 -26396.074} C_VEL
LIN {X 0,Y 117.572,Z 837.199,A -85,B 0,C 180,E1 -26402.542,E2 -26402.542} C_VEL
LIN {X 0,Y 124.685,Z 834.485,A -85,B 0,C 180,E1 -26408.313,E2 -26408.313} C_VEL
LIN {X 0,Y 130.904,Z 831.445,A -85,B 0,C 180,E1 -26412.147,E2 -26412.147} C_VEL
LIN {X 0,Y 137.889,Z 827.485,A -85,B 0,C 180,E1 -26415.52,E2 -26415.52} C_VEL
LIN {X 0,Y 145.289,Z 822.596,A -85,B 0,C 180,E1 -26418.566,E2 -26418.566} C_VEL
LIN {X 0,Y 154.554,Z 815.484,A -85,B 0,C 180,E1 -26421.661,E2 -26421.661} C_VEL
LIN {X 0,Y 162.928,Z 807.92,A -85,B 0,C 180,E1 -26423.973,E2 -26423.973} C_VEL
LIN {X 0,Y 171.705,Z 798.72,A -85,B 0,C 180,E1 -26425.975,E2 -26425.975} C_VEL
LIN {X 0,Y 175.416,Z 794.335,A -85,B 0,C 180,E1 -26426.721,E2 -26426.721} C_VEL
LIN {X 0,Y 178.635,Z 790.123,A -85,B 0,C 180,E1 -26427.569,E2 -26427.569} C_VEL
LIN {X 0,Y 183.209,Z 783.295,A -85,B 0,C 180,E1 -26429.334,E2 -26429.334} C_VEL
LIN {X 0,Y 187.529,Z 776.081,A -85,B 0,C 180,E1 -26430.922,E2 -26430.922} C_VEL
LIN {X 0,Y 190.257,Z 771.261,A -85,B 0,C 180,E1 -26431.509,E2 -26431.509} C_VEL
LIN {X 0,Y 196.766,Z 758.372,A -85,B 0,C 180,E1 -26432.333,E2 -26432.333} C_VEL
LIN {X 0,Y 201.406,Z 746.612,A -85,B 0,C 180,E1 -26432.837,E2 -26432.837} C_VEL
LIN {X 0,Y 201.967,Z 744.83,A -85,B 0,C 180,E1 -26433.104,E2 -26433.104} C_VEL
LIN {X 0,Y 196.851,Z 757.927,A -85,B 0,C 180,E1 -26433.95,E2 -26433.95} C_VEL
LIN {X 0,Y 190.909,Z 769.601,A -85,B 0,C 180,E1 -26434.953,E2 -26434.953} C_VEL
LIN {X 0,Y 183.699,Z 780.978,A -85,B 0,C 180,E1 -26436.243,E2 -26436.243} C_VEL
LIN {X 0,Y 175.415,Z 791.52,A -85,B 0,C 180,E1 -26437.886,E2 -26437.886} C_VEL
LIN {X 0,Y 167.191,Z 800.331,A -85,B 0,C 180,E1 -26439.708,E2 -26439.708} C_VEL
LIN {X 0,Y 158.555,Z 808.065,A -85,B 0,C 180,E1 -26441.924,E2 -26441.924} C_VEL
LIN {X 0,Y 148.485,Z 815.438,A -85,B 0,C 180,E1 -26444.91,E2 -26444.91} C_VEL
LIN {X 0,Y 139.069,Z 821.118,A -85,B 0,C 180,E1 -26448.337,E2 -26448.337} C_VEL
LIN {X 0,Y 130.294,Z 825.245,A -85,B 0,C 180,E1 -26452.25,E2 -26452.25} C_VEL
LIN {X 0,Y 122.314,Z 828.049,A -85,B 0,C 180,E1 -26456.706,E2 -26456.706} C_VEL
LIN {X 0,Y 117.508,Z 829.256,A -85,B 0,C 180,E1 -26460,E2 -26460} C_VEL
LIN {X 0,Y 112.713,Z 829.946,A -85,B 0,C 180,E1 -26463.99,E2 -26463.99} C_VEL
LIN {X 0,Y 107.066,Z 829.868,A -85,B 0,C 180,E1 -26470.085,E2 -26470.085} C_VEL
LIN {X 0,Y 102.719,Z 828.577,A -85,B 0,C 180,E1 -26476.705,E2 -26476.705} C_VEL
LIN {X 0,Y 99.765,Z 826.084,A -85,B 0,C 180,E1 -26483.693,E2 -26483.693} C_VEL
LIN {X 0,Y 98.278,Z 822.336,A -85,B 0,C 180,E1 -26490.901,E2 -26490.901} C_VEL
LIN {X 0,Y 98.133,Z 817.295,A -85,B 0,C 180,E1 -26498.029,E2 -26498.029} C_VEL
LIN {X 0,Y 99.013,Z 811.049,A -85,B 0,C 180,E1 -26504.788,E2 -26504.788} C_VEL
LIN {X 0,Y 100.573,Z 803.634,A -85,B 0,C 180,E1 -26511.036,E2 -26511.036} C_VEL
LIN {X 0,Y 102.915,Z 794.636,A -85,B 0,C 180,E1 -26516.891,E2 -26516.891} C_VEL
LIN {X 0,Y 105.956,Z 784.274,A -85,B 0,C 180,E1 -26522.105,E2 -26522.105} C_VEL
LIN {X 0,Y 108.674,Z 774.535,A -85,B 0,C 180,E1 -26525.888,E2 -26525.888} C_VEL
LIN {X 0,Y 111.943,Z 762.182,A -85,B 0,C 180,E1 -26529.556,E2 -26529.556} C_VEL
LIN {X 0,Y 114.518,Z 750.741,A -85,B 0,C 180,E1 -26532.135,E2 -26532.135} C_VEL
LIN {X 0,Y 116.95,Z 737.322,A -85,B 0,C 180,E1 -26534.336,E2 -26534.336} C_VEL
LIN {X 0,Y 118.647,Z 724.119,A -85,B 0,C 180,E1 -26535.852,E2 -26535.852} C_VEL
LIN {X 0,Y 122.586,Z 679.774,A -85,B 0,C 180,E1 -26539.014,E2 -26539.014} C_VEL
LIN {X 0,Y 114.986,Z 660.756,A -85,B 0,C 180,E1 -26542.886,E2 -26542.886} C_VEL
LIN {X 0,Y 108.978,Z 647.521,A -85,B 0,C 180,E1 -26546.152,E2 -26546.152} C_VEL
LIN {X 0,Y 101.879,Z 633.318,A -85,B 0,C 180,E1 -26550.498,E2 -26550.498} C_VEL
LIN {X 0,Y 101.764,Z 632.811,A -85,B 0,C 180,E1 -26550.746,E2 -26550.746} C_VEL
LIN {X 0,Y 101.281,Z 632.868,A -85,B 0,C 180,E1 -26557.982,E2 -26557.982} C_VEL
LIN {X 0,Y 101.131,Z 632.888,A -85,B 0,C 180,E1 -26563.367,E2 -26563.367} C_VEL
LIN {X 0,Y 100.819,Z 632.903,A -85,B 0,C 180,E1 -26570.403,E2 -26570.403} C_VEL
LIN {X 0,Y 100.777,Z 632.931,A -85,B 0,C 180,E1 -26574.962,E2 -26574.962} C_VEL
LIN {X 0,Y 100.695,Z 632.903,A -85,B 0,C 180,E1 -26583.12,E2 -26583.12} C_VEL
LIN {X 0,Y 100.645,Z 632.941,A -85,B 0,C 180,E1 -26589.815,E2 -26589.815} C_VEL
LIN {X 0,Y 100.653,Z 632.937,A -85,B 0,C 180,E1 -26595.714,E2 -26595.714} C_VEL
LIN {X 0,Y 100.636,Z 632.898,A -85,B 0,C 180,E1 -26601.059,E2 -26601.059} C_VEL
LIN {X 0,Y 100.7,Z 632.916,A -85,B 0,C 180,E1 -26606.884,E2 -26606.884} C_VEL
LIN {X 0,Y 100.793,Z 632.927,A -85,B 0,C 180,E1 -26615.269,E2 -26615.269} C_VEL
LIN {X 0,Y 100.817,Z 632.9,A -85,B 0,C 180,E1 -26619.602,E2 -26619.602} C_VEL
LIN {X 0,Y 101.166,Z 632.862,A -85,B 0,C 180,E1 -26627.971,E2 -26627.971} C_VEL
LIN {X 0,Y 101.25,Z 632.87,A -85,B 0,C 180,E1 -26632.021,E2 -26632.021} C_VEL
LIN {X 0,Y 101.854,Z 632.767,A -85,B 0,C 180,E1 -26640.001,E2 -26640.001} C_VEL
LIN {X 0,Y 101.243,Z 632.872,A -85,B 0,C 180,E1 -26647.981,E2 -26647.981} C_VEL
LIN {X 0,Y 101.062,Z 632.883,A -85,B 0,C 180,E1 -26653.182,E2 -26653.182} C_VEL
LIN {X 0,Y 100.81,Z 632.932,A -85,B 0,C 180,E1 -26660.401,E2 -26660.401} C_VEL
LIN {X 0,Y 100.782,Z 632.921,A -85,B 0,C 180,E1 -26664.957,E2 -26664.957} C_VEL
LIN {X 0,Y 100.758,Z 633.092,A -85,B 0,C 180,E1 -26672.765,E2 -26672.765} C_VEL
LIN {X 0,Y 101.768,Z 635.847,A -85,B 0,C 180,E1 -26673.537,E2 -26673.537} C_VEL
LIN {X 0,Y 102.983,Z 637.72,A -85,B 0,C 180,E1 -26674.265,E2 -26674.265} C_VEL
LIN {X 0,Y 108.86,Z 648.383,A -85,B 0,C 180,E1 -26677.667,E2 -26677.667} C_VEL
LIN {X 0,Y 114.718,Z 664.168,A -85,B 0,C 180,E1 -26681.156,E2 -26681.156} C_VEL
LIN {X 0,Y 120.525,Z 682.795,A -85,B 0,C 180,E1 -26684.528,E2 -26684.528} C_VEL
LIN {X 0,Y 121.6,Z 701.225,A -85,B 0,C 180,E1 -26686.458,E2 -26686.458} C_VEL
LIN {X 0,Y 118.138,Z 739.14,A -85,B 0,C 180,E1 -26689.263,E2 -26689.263} C_VEL
LIN {X 0,Y 116.225,Z 752.382,A -85,B 0,C 180,E1 -26690.861,E2 -26690.861} C_VEL
LIN {X 0,Y 113.661,Z 764.94,A -85,B 0,C 180,E1 -26693.031,E2 -26693.031} C_VEL
LIN {X 0,Y 110.509,Z 777.697,A -85,B 0,C 180,E1 -26696.082,E2 -26696.082} C_VEL
LIN {X 0,Y 107.531,Z 788.55,A -85,B 0,C 180,E1 -26699.563,E2 -26699.563} C_VEL
LIN {X 0,Y 104.543,Z 799.253,A -85,B 0,C 180,E1 -26704.085,E2 -26704.085} C_VEL
LIN {X 0,Y 102.163,Z 807.974,A -85,B 0,C 180,E1 -26708.824,E2 -26708.824} C_VEL
LIN {X 0,Y 100.498,Z 815.178,A -85,B 0,C 180,E1 -26713.752,E2 -26713.752} C_VEL
LIN {X 0,Y 99.363,Z 822.153,A -85,B 0,C 180,E1 -26719.811,E2 -26719.811} C_VEL
LIN {X 0,Y 99.177,Z 827.664,A -85,B 0,C 180,E1 -26725.932,E2 -26725.932} C_VEL
LIN {X 0,Y 99.179,Z 830.559,A -85,B 0,C 180,E1 -26729.996,E2 -26729.996} C_VEL
LIN {X 0,Y 98.899,Z 833.677,A -85,B 0,C 180,E1 -26735.796,E2 -26735.796} C_VEL
LIN {X 0,Y 99.167,Z 836.087,A -85,B 0,C 180,E1 -26742.271,E2 -26742.271} C_VEL
LIN {X 0,Y 101.282,Z 837.781,A -85,B 0,C 180,E1 -26750.296,E2 -26750.296} C_VEL
LIN {X 0,Y 105.572,Z 838.128,A -85,B 0,C 180,E1 -26757.77,E2 -26757.77} C_VEL
LIN {X 0,Y 111.626,Z 837.077,A -85,B 0,C 180,E1 -26764.511,E2 -26764.511} C_VEL
LIN {X 0,Y 119.193,Z 834.622,A -85,B 0,C 180,E1 -26770.431,E2 -26770.431} C_VEL
LIN {X 0,Y 128.087,Z 830.742,A -85,B 0,C 180,E1 -26775.499,E2 -26775.499} C_VEL
LIN {X 0,Y 135.501,Z 826.784,A -85,B 0,C 180,E1 -26778.764,E2 -26778.764} C_VEL
LIN {X 0,Y 143.432,Z 821.829,A -85,B 0,C 180,E1 -26781.621,E2 -26781.621} C_VEL
LIN {X 0,Y 153.168,Z 814.697,A -85,B 0,C 180,E1 -26784.527,E2 -26784.527} C_VEL
LIN {X 0,Y 161.9,Z 807.149,A -85,B 0,C 180,E1 -26786.676,E2 -26786.676} C_VEL
LIN {X 0,Y 171.013,Z 797.838,A -85,B 0,C 180,E1 -26788.506,E2 -26788.506} C_VEL
LIN {X 0,Y 180.333,Z 786.482,A -85,B 0,C 180,E1 -26790.122,E2 -26790.122} C_VEL
LIN {X 0,Y 188.332,Z 774.533,A -85,B 0,C 180,E1 -26791.271,E2 -26791.271} C_VEL
